# B&R Automation Studio project NAEUL004C00R13L518F00 (part 10)

#### Act_Main_P0933.st
```iecst
ACTION Act_Main_P0933:

	//Display
	tyP0933PushConv.tyFB.tyNumExtSpd.uiRtStat.0			:= NOT p_tyNtParamCurr.bProjMotorizedPusherPrep;
	tyP0933PushConv.tyFB.tyNumExtTorqPercent.uiRtStat.0	:= NOT p_tyNtParamCurr.bProjMotorizedPusherPrep;

	tyP0933PushConv.tyDC.tyBtnSpdBinBit0.uiRtStat.0	:=  NOT p_tyNtParamCurr.bProjMotorizedPusherPrep;
	tyP0933PushConv.tyDC.tyBtnSpdBinBit1.uiRtStat.0	:=  NOT p_tyNtParamCurr.bProjMotorizedPusherPrep;
	tyP0933PushConv.tyDC.tyBtnSpdBinBit2.uiRtStat.0	:=  NOT p_tyNtParamCurr.bProjMotorizedPusherPrep;

	tyP0933PushConv.tyDC.tyBtnSigOn.uiRtStat.0	:=  NOT p_tyNtParamCurr.bProjMotorizedPusherPrep;
	tyP0933PushConv.tyDC.tyBtnAlarmRst.uiRtStat.0:=  NOT p_tyNtParamCurr.bProjMotorizedPusherPrep;

	//Display
	tyP0933PushConv.tyFB.tyNumExtSpd.diValueMin	:= p_tyNtParamCurr.tyProdRcpMtrPshrExtSpd.diMin;
	tyP0933PushConv.tyFB.tyNumExtSpd.diValueMax	:= p_tyNtParamCurr.tyProdRcpMtrPshrExtSpd.diMax;

	tyP0933PushConv.tyFB.tyNumExtTorqPercent.diValueMin	:= p_tyNtParamCurr.tyProdRcpMtrPshrExtTorq.diMin;
	tyP0933PushConv.tyFB.tyNumExtTorqPercent.diValueMax	:= p_tyNtParamCurr.tyProdRcpMtrPshrExtTorq.diMax;

	tyP0933PushConv.tyCom.tyBtnExtSlwSen.uiRtStat.0 := NOT p_tyNtParamCurr.bProjMotorizedPusherPrep;
	tyP0933PushConv.tyCom.tyBtnRetSlwSen.uiRtStat.0 := NOT p_tyNtParamCurr.bProjMotorizedPusherPrep;
	tyP0933PushConv.tyCom.tyBtnAlarmSig.uiRtStat.0 := NOT p_tyNtParamCurr.bProjMotorizedPusherPrep;
	tyP0933PushConv.tyCom.tyBtnTorqueSig.uiRtStat.0 := NOT p_tyNtParamCurr.bProjMotorizedPusherPrep;

	tyP0933PushConv.tyDC.tyBtnAlarmRst.uiRtStat.0 := NOT p_tyNtParamCurr.bProjMotorizedPusherPrep;
	tyP0933PushConv.tyDC.tyBtnSigOn.uiRtStat.0 := NOT p_tyNtParamCurr.bProjMotorizedPusherPrep;

	tyP0933PushConv.tyCom.tyBtnAntiJamSen.uiRtStat.0 := p_tyNtParamCurr.tyDISettings.diPshrAntiJam = 0;
	tyP0933PushConv.tyCom.tyBtnAlarmSig.uiRtStat.0	 := p_tyNtParamCurr.tyDISettings.diMtrPshrAlmSig = 0;
	tyP0933PushConv.tyCom.tyBtnTorqueSig.uiRtStat.0  := p_tyNtParamCurr.tyDISettings.diMtrPshrTorqueSig = 0;

END_ACTION
```

#### Act_Main_P0934.st
```iecst
ACTION Act_Main_P0934:

	//Display
	tyP0934AW.tyMotionStd.tyNumTargetPos.diValue	:= 0;
	tyP0934AW.tyMotionStd.tyNumStepSize.diValue		:= 0;
	tyP0934AW.tyMotionStd.tyNumNomSpd.diValue		:= (p_tyNtParamCurr.tyUIAWNomSpd.diMax + p_tyNtParamCurr.tyUIAWNomSpd.diMin) / 2;
	tyP0934AW.tyMotionStd.tyNumSlwSpd.diValue		:= (p_tyNtParamCurr.tyUIAWSlwSpd.diMax + p_tyNtParamCurr.tyUIAWSlwSpd.diMin) / 3;

	tyP0934AW.tyMotionStd.tyNumTargetPos.diValueMax	:= p_tyNtParamCurr.tyProdRcpWidth.diMax;
	tyP0934AW.tyMotionStd.tyNumTargetPos.diValueMin	:= p_tyNtParamCurr.tyUIAWTargetPos.diMin;

	tyP0934AW.tyMotionStd.tyNumStepSize.diValueMax	:= p_tyNtParamCurr.tyProdRcpWidth.diMax;
	tyP0934AW.tyMotionStd.tyNumStepSize.diValueMin	:= p_tyNtParamCurr.tyProdRcpWidth.diMax * -1;

	tyP0934AW.tyMotionStd.tyNumNomSpd.diValueMax	:= p_tyNtParamCurr.tyUIAWNomSpd.diMax;
	tyP0934AW.tyMotionStd.tyNumNomSpd.diValueMin	:= p_tyNtParamCurr.tyUIAWNomSpd.diMin;

	tyP0934AW.tyMotionStd.tyNumSlwSpd.diValueMax	:= p_tyNtParamCurr.tyUIAWSlwSpd.diMax;
	tyP0934AW.tyMotionStd.tyNumSlwSpd.diValueMin	:= p_tyNtParamCurr.tyUIAWSlwSpd.diMin;

	tyP0934AW.tyAW.tyNumNewWidth.diValueMax			:= p_tyNtParamCurr.tyProdRcpWidth.diMax;
	tyP0934AW.tyAW.tyNumNewWidth.diValueMin			:= p_tyNtParamCurr.tyProdRcpWidth.diMin;

END_ACTION
```

#### Act_Main_P0935.st
```iecst
ACTION Act_Main_P0935:

	tyP0935Lifter.tyLifter.tyBtnGoLaneB.uiRtStat.0	:= NOT p_tyNtParamCurr.bProjLaneBPrep;
	tyP0935Lifter.tyLifter.tyBtnGoLaneA.uiRtStat 		:= p_tyNtParamCurr.bProjMagConvLane1Prep;
	tyP0935Lifter.tyLifter.tyBtnGoLaneA.uiMaskRtStat 	:= p_tyNtParamCurr.bProjMagConvLane1Prep;
	tyP0935Lifter.tyLifter.tyBtnGoLaneD_G.uiRtStat 		:= NOT (p_tyNtParamCurr.bProjMagConvLane1Prep);
	tyP0935Lifter.tyLifter.tyBtnGoLaneD_G.uiMaskRtStat 	:= NOT (p_tyNtParamCurr.bProjMagConvLane1Prep);
	tyP0935Lifter.tyLifter.tyBtnGoLaneE_H.uiRtStat 		:= NOT (p_tyNtParamCurr.bProjMagConvLane1Prep);
	tyP0935Lifter.tyLifter.tyBtnGoLaneE_H.uiMaskRtStat 	:= NOT (p_tyNtParamCurr.bProjMagConvLane1Prep);

	//Display
	tyP0935Lifter.tyMotionStd.tyNumTargetPos.diValue	:= 0;
	tyP0935Lifter.tyMotionStd.tyNumStepSize.diValue		:= 0;
	tyP0935Lifter.tyMotionStd.tyNumNomSpd.diValue		:= (p_tyNtParamCurr.tyUILifterNomSpd.diMax + p_tyNtParamCurr.tyUILifterNomSpd.diMin) / 2;
	tyP0935Lifter.tyMotionStd.tyNumSlwSpd.diValue		:= (p_tyNtParamCurr.tyUILifterSlwSpd.diMax + p_tyNtParamCurr.tyUILifterSlwSpd.diMin) / 3;

	tyP0935Lifter.tyMotionStd.tyNumTargetPos.diValueMax	:= p_tyNtParamCurr.tyUILifterTargetPos.diMax;
	tyP0935Lifter.tyMotionStd.tyNumTargetPos.diValueMin	:= p_tyNtParamCurr.tyUILifterTargetPos.diMin;

	tyP0935Lifter.tyMotionStd.tyNumStepSize.diValueMax	:= p_tyNtParamCurr.tyUILifterStepSize.diMax;
	tyP0935Lifter.tyMotionStd.tyNumStepSize.diValueMin	:= p_tyNtParamCurr.tyUILifterStepSize.diMin;

	tyP0935Lifter.tyMotionStd.tyNumNomSpd.diValueMax	:= p_tyNtParamCurr.tyUILifterNomSpd.diMax;
	tyP0935Lifter.tyMotionStd.tyNumNomSpd.diValueMin	:= p_tyNtParamCurr.tyUILifterNomSpd.diMin;

	tyP0935Lifter.tyMotionStd.tyNumSlwSpd.diValueMax	:= p_tyNtParamCurr.tyUILifterSlwSpd.diMax;
	tyP0935Lifter.tyMotionStd.tyNumSlwSpd.diValueMin	:= p_tyNtParamCurr.tyUILifterSlwSpd.diMin;

	tyP0935Lifter.tyLifter.tyNumMagPos.diValue			:= 1;
	tyP0935Lifter.tyLifter.tyNumMagPos.diValueMin		:= 1;

	CASE p_tyNtParamCurr.eProjMag OF

		ULMagDual:
			IF p_tyNtParamCurr.bProjMagConvLane1Prep THEN
				tyP0935Lifter.tyLifter.tyNumMagPos.diValueMax		:= 1;
			ELSE
				tyP0935Lifter.tyLifter.tyNumMagPos.diValueMax		:= 2;
			END_IF

		ULMagTriple:
			tyP0935Lifter.tyLifter.tyNumMagPos.diValueMax		:= 3;

		ULMagQuadruple:
			tyP0935Lifter.tyLifter.tyNumMagPos.diValueMax		:= 4;

	END_CASE

	IF p_tyNtParamCurr.bProjLifterMagPlatform THEN
		tyP0935Lifter.tyLifter.tyBtnGoLaneA.usiTxtIdx := 23;
	END_IF

END_ACTION
```

#### Act_Main_P0936.st
```iecst
ACTION Act_Main_P0936:

	//Display
	tyP0936Trav.tyTrav.tyBtnGoToLaneB.uiRtStat.0	:= NOT p_tyNtParamCurr.bProjLaneBPrep;
	tyP0936Trav.tyTrav.tyBtnGoToMag3.uiRtStat.0		:= NOT(p_tyNtParamCurr.eProjMag = ULMagTriple);

	tyP0936Trav.tyMotionStd.tyNumTargetPos.diValue		:= 0;
	tyP0936Trav.tyMotionStd.tyNumStepSize.diValue		:= 0;
	tyP0936Trav.tyMotionStd.tyNumNomSpd.diValue			:= (p_tyNtParamCurr.tyUITravNomSpd.diMax + p_tyNtParamCurr.tyUITravNomSpd.diMin) / 2;
	tyP0936Trav.tyMotionStd.tyNumSlwSpd.diValue			:= (p_tyNtParamCurr.tyUITravSlwSpd.diMax + p_tyNtParamCurr.tyUITravSlwSpd.diMin) / 3;

	tyP0936Trav.tyMotionStd.tyNumTargetPos.diValueMax	:= p_tyNtParamCurr.tyUITravTargetPos.diMax;
	tyP0936Trav.tyMotionStd.tyNumTargetPos.diValueMin	:= p_tyNtParamCurr.tyUITravTargetPos.diMin;

	tyP0936Trav.tyMotionStd.tyNumStepSize.diValueMax	:= p_tyNtParamCurr.tyUITravStepSize.diMax;
	tyP0936Trav.tyMotionStd.tyNumStepSize.diValueMin	:= p_tyNtParamCurr.tyUITravStepSize.diMin;

	tyP0936Trav.tyMotionStd.tyNumNomSpd.diValueMax		:= p_tyNtParamCurr.tyUITravNomSpd.diMax;
	tyP0936Trav.tyMotionStd.tyNumNomSpd.diValueMin		:= p_tyNtParamCurr.tyUITravNomSpd.diMin;

	tyP0936Trav.tyMotionStd.tyNumSlwSpd.diValueMax		:= p_tyNtParamCurr.tyUITravSlwSpd.diMax;
	tyP0936Trav.tyMotionStd.tyNumSlwSpd.diValueMin		:= p_tyNtParamCurr.tyUITravSlwSpd.diMin;

END_ACTION
```

#### Act_Main_P0937.st
```iecst
ACTION Act_Main_P0937:

	//Display
	tyP0937AWPushOrPuller.tyMotionStd.tyNumTargetPos.diValue	:= 0;
	tyP0937AWPushOrPuller.tyMotionStd.tyNumStepSize.diValue		:= 0;
	tyP0937AWPushOrPuller.tyMotionStd.tyNumNomSpd.diValue		:= (p_tyNtParamCurr.tyUIAWNomSpd.diMax + p_tyNtParamCurr.tyUIAWNomSpd.diMin) / 2;
	tyP0937AWPushOrPuller.tyMotionStd.tyNumSlwSpd.diValue		:= (p_tyNtParamCurr.tyUIAWSlwSpd.diMax + p_tyNtParamCurr.tyUIAWSlwSpd.diMin) / 3;

	tyP0937AWPushOrPuller.tyMotionStd.tyNumTargetPos.diValueMax	:= p_tyNtParamCurr.tyProdRcpWidth.diMax;
	tyP0937AWPushOrPuller.tyMotionStd.tyNumTargetPos.diValueMin	:= p_tyNtParamCurr.tyUIAWTargetPos.diMin;

	tyP0937AWPushOrPuller.tyMotionStd.tyNumStepSize.diValueMax	:= p_tyNtParamCurr.tyProdRcpWidth.diMax;
	tyP0937AWPushOrPuller.tyMotionStd.tyNumStepSize.diValueMin	:= p_tyNtParamCurr.tyProdRcpWidth.diMax * -1;

	tyP0937AWPushOrPuller.tyMotionStd.tyNumNomSpd.diValueMax	:= p_tyNtParamCurr.tyUIAWNomSpd.diMax;
	tyP0937AWPushOrPuller.tyMotionStd.tyNumNomSpd.diValueMin	:= p_tyNtParamCurr.tyUIAWNomSpd.diMin;

	tyP0937AWPushOrPuller.tyMotionStd.tyNumSlwSpd.diValueMax	:= p_tyNtParamCurr.tyUIAWSlwSpd.diMax;
	tyP0937AWPushOrPuller.tyMotionStd.tyNumSlwSpd.diValueMin	:= p_tyNtParamCurr.tyUIAWSlwSpd.diMin;

	tyP0937AWPushOrPuller.tyAW.tyNumNewWidth.diValueMax			:= p_tyNtParamCurr.tyProdRcpWidth.diMax;
	tyP0937AWPushOrPuller.tyAW.tyNumNewWidth.diValueMin			:= p_tyNtParamCurr.tyProdRcpWidth.diMin;

END_ACTION
```

#### Act_Main_P0938.st
```iecst
ACTION Act_Main_P0938:

	//Display
	//Magazine Auto Width 1
	tyP0938MagAW.tyMotionStd1.tyNumTargetPos.diValue	:= 0;
	tyP0938MagAW.tyMotionStd1.tyNumStepSize.diValue		:= 0;
	tyP0938MagAW.tyMotionStd1.tyNumNomSpd.diValue		:= (p_tyNtParamCurr.tyUIMagAWNomSpd.diMax + p_tyNtParamCurr.tyUIMagAWNomSpd.diMin) / 2;
	tyP0938MagAW.tyMotionStd1.tyNumSlwSpd.diValue		:= (p_tyNtParamCurr.tyUIMagAWSlwSpd.diMax + p_tyNtParamCurr.tyUIMagAWSlwSpd.diMin) / 3;

	tyP0938MagAW.tyMotionStd1.tyNumTargetPos.diValueMax	:= p_tyNtParamCurr.tyProdRcpWidth.diMax;
	tyP0938MagAW.tyMotionStd1.tyNumTargetPos.diValueMin	:= p_tyNtParamCurr.tyUIMagAWTargetPos.diMin;

	tyP0938MagAW.tyMotionStd1.tyNumStepSize.diValueMax	:= p_tyNtParamCurr.tyProdRcpWidth.diMax;
	tyP0938MagAW.tyMotionStd1.tyNumStepSize.diValueMin	:= p_tyNtParamCurr.tyProdRcpWidth.diMax * -1;

	tyP0938MagAW.tyMotionStd1.tyNumNomSpd.diValueMax	:= p_tyNtParamCurr.tyUIMagAWNomSpd.diMax;
	tyP0938MagAW.tyMotionStd1.tyNumNomSpd.diValueMin	:= p_tyNtParamCurr.tyUIMagAWNomSpd.diMin;

	tyP0938MagAW.tyMotionStd1.tyNumSlwSpd.diValueMax	:= p_tyNtParamCurr.tyUIMagAWSlwSpd.diMax;
	tyP0938MagAW.tyMotionStd1.tyNumSlwSpd.diValueMin	:= p_tyNtParamCurr.tyUIMagAWSlwSpd.diMin;

	tyP0938MagAW.tyMagAW1.tyNumNewWidth.diValueMax		:= p_tyNtParamCurr.tyProdRcpWidth.diMax;
	tyP0938MagAW.tyMagAW1.tyNumNewWidth.diValueMin		:= p_tyNtParamCurr.tyProdRcpWidth.diMin;

	//Magazine Auto Width 2
	tyP0938MagAW.tyMotionStd2.tyNumTargetPos.diValue	:= 0;
	tyP0938MagAW.tyMotionStd2.tyNumStepSize.diValue		:= 0;
	tyP0938MagAW.tyMotionStd2.tyNumNomSpd.diValue		:= (p_tyNtParamCurr.tyUIMagAWNomSpd.diMax + p_tyNtParamCurr.tyUIMagAWNomSpd.diMin) / 2;
	tyP0938MagAW.tyMotionStd2.tyNumSlwSpd.diValue		:= (p_tyNtParamCurr.tyUIMagAWSlwSpd.diMax + p_tyNtParamCurr.tyUIMagAWSlwSpd.diMin) / 3;

	tyP0938MagAW.tyMotionStd2.tyNumTargetPos.diValueMax	:= p_tyNtParamCurr.tyProdRcpWidth.diMax;
	tyP0938MagAW.tyMotionStd2.tyNumTargetPos.diValueMin	:= p_tyNtParamCurr.tyUIMagAWTargetPos.diMin;

	tyP0938MagAW.tyMotionStd2.tyNumStepSize.diValueMax	:= p_tyNtParamCurr.tyProdRcpWidth.diMax;
	tyP0938MagAW.tyMotionStd2.tyNumStepSize.diValueMin	:= p_tyNtParamCurr.tyProdRcpWidth.diMax * -1;

	tyP0938MagAW.tyMotionStd2.tyNumNomSpd.diValueMax	:= p_tyNtParamCurr.tyUIMagAWNomSpd.diMax;
	tyP0938MagAW.tyMotionStd2.tyNumNomSpd.diValueMin	:= p_tyNtParamCurr.tyUIMagAWNomSpd.diMin;

	tyP0938MagAW.tyMotionStd2.tyNumSlwSpd.diValueMax	:= p_tyNtParamCurr.tyUIMagAWSlwSpd.diMax;
	tyP0938MagAW.tyMotionStd2.tyNumSlwSpd.diValueMin	:= p_tyNtParamCurr.tyUIMagAWSlwSpd.diMin;

	tyP0938MagAW.tyMagAW2.tyNumNewWidth.diValueMax		:= p_tyNtParamCurr.tyProdRcpWidth.diMax;
	tyP0938MagAW.tyMagAW2.tyNumNewWidth.diValueMin		:= p_tyNtParamCurr.tyProdRcpWidth.diMin;

	//Magazine Auto Width 3
	tyP0938MagAW.tyMotionStd3.tyNumTargetPos.diValue	:= 0;
	tyP0938MagAW.tyMotionStd3.tyNumStepSize.diValue		:= 0;
	tyP0938MagAW.tyMotionStd3.tyNumNomSpd.diValue		:= (p_tyNtParamCurr.tyUIMagAWNomSpd.diMax + p_tyNtParamCurr.tyUIMagAWNomSpd.diMin) / 2;
	tyP0938MagAW.tyMotionStd3.tyNumSlwSpd.diValue		:= (p_tyNtParamCurr.tyUIMagAWSlwSpd.diMax + p_tyNtParamCurr.tyUIMagAWSlwSpd.diMin) / 3;

	tyP0938MagAW.tyMotionStd3.tyNumTargetPos.diValueMax	:= p_tyNtParamCurr.tyProdRcpWidth.diMax;
	tyP0938MagAW.tyMotionStd3.tyNumTargetPos.diValueMin	:= p_tyNtParamCurr.tyUIMagAWTargetPos.diMin;

	tyP0938MagAW.tyMotionStd3.tyNumStepSize.diValueMax	:= p_tyNtParamCurr.tyProdRcpWidth.diMax;
	tyP0938MagAW.tyMotionStd3.tyNumStepSize.diValueMin	:= p_tyNtParamCurr.tyProdRcpWidth.diMax * -1;

	tyP0938MagAW.tyMotionStd3.tyNumNomSpd.diValueMax	:= p_tyNtParamCurr.tyUIMagAWNomSpd.diMax;
	tyP0938MagAW.tyMotionStd3.tyNumNomSpd.diValueMin	:= p_tyNtParamCurr.tyUIMagAWNomSpd.diMin;

	tyP0938MagAW.tyMotionStd3.tyNumSlwSpd.diValueMax	:= p_tyNtParamCurr.tyUIMagAWSlwSpd.diMax;
	tyP0938MagAW.tyMotionStd3.tyNumSlwSpd.diValueMin	:= p_tyNtParamCurr.tyUIMagAWSlwSpd.diMin;

	tyP0938MagAW.tyMagAW3.tyNumNewWidth.diValueMax		:= p_tyNtParamCurr.tyProdRcpWidth.diMax;
	tyP0938MagAW.tyMagAW3.tyNumNewWidth.diValueMin		:= p_tyNtParamCurr.tyProdRcpWidth.diMin;

END_ACTION
```

#### Act_Main_P0939.st
```iecst
ACTION Act_Main_P0939:

	tyP0939Lifter2.tyLifter.tyBtnGoLaneB.uiRtStat.0	:= NOT p_tyNtParamCurr.bProjLaneBPrep;
	tyP0939Lifter2.tyLifter.tyBtnGoLaneA.uiRtStat.0	:= p_tyNtParamCurr.bProjMagConvLane2Prep;
	tyP0939Lifter2.tyLifter.tyBtnGoLaneA.uiRtStat.0	:= p_tyNtParamCurr.bProjMagConvLane2Prep;
	tyP0935Lifter.tyLifter.tyBtnGoLaneD_G.uiRtStat 		:= NOT (p_tyNtParamCurr.bProjMagConvLane2Prep);
	tyP0935Lifter.tyLifter.tyBtnGoLaneD_G.uiMaskRtStat 	:= NOT (p_tyNtParamCurr.bProjMagConvLane2Prep);
	tyP0935Lifter.tyLifter.tyBtnGoLaneE_H.uiRtStat 		:= NOT (p_tyNtParamCurr.bProjMagConvLane2Prep);
	tyP0935Lifter.tyLifter.tyBtnGoLaneE_H.uiMaskRtStat 	:= NOT (p_tyNtParamCurr.bProjMagConvLane2Prep);

	//Display
	tyP0939Lifter2.tyMotionStd.tyNumTargetPos.diValue	:= 0;
	tyP0939Lifter2.tyMotionStd.tyNumStepSize.diValue		:= 0;
	tyP0939Lifter2.tyMotionStd.tyNumNomSpd.diValue		:= (p_tyNtParamCurr.tyUILifterNomSpd.diMax + p_tyNtParamCurr.tyUILifterNomSpd.diMin) / 2;
	tyP0939Lifter2.tyMotionStd.tyNumSlwSpd.diValue		:= (p_tyNtParamCurr.tyUILifterSlwSpd.diMax + p_tyNtParamCurr.tyUILifterSlwSpd.diMin) / 3;

	tyP0939Lifter2.tyMotionStd.tyNumTargetPos.diValueMax	:= p_tyNtParamCurr.tyUILifterTargetPos.diMax;
	tyP0939Lifter2.tyMotionStd.tyNumTargetPos.diValueMin	:= p_tyNtParamCurr.tyUILifterTargetPos.diMin;

	tyP0939Lifter2.tyMotionStd.tyNumStepSize.diValueMax	:= p_tyNtParamCurr.tyUILifterStepSize.diMax;
	tyP0939Lifter2.tyMotionStd.tyNumStepSize.diValueMin	:= p_tyNtParamCurr.tyUILifterStepSize.diMin;

	tyP0939Lifter2.tyMotionStd.tyNumNomSpd.diValueMax	:= p_tyNtParamCurr.tyUILifterNomSpd.diMax;
	tyP0939Lifter2.tyMotionStd.tyNumNomSpd.diValueMin	:= p_tyNtParamCurr.tyUILifterNomSpd.diMin;

	tyP0939Lifter2.tyMotionStd.tyNumSlwSpd.diValueMax	:= p_tyNtParamCurr.tyUILifterSlwSpd.diMax;
	tyP0939Lifter2.tyMotionStd.tyNumSlwSpd.diValueMin	:= p_tyNtParamCurr.tyUILifterSlwSpd.diMin;

	tyP0939Lifter2.tyLifter.tyNumMagPos.diValue			:= 2;
	tyP0939Lifter2.tyLifter.tyNumMagPos.diValueMin		:= 2;
	tyP0939Lifter2.tyLifter.tyNumMagPos.diValueMax		:= 2;

	CASE p_tyNtParamCurr.eProjMag OF

		ULMagDual:
			tyP0939Lifter2.tyLifter.tyNumMagPos.diValueMax		:= 2;

		ULMagTriple:
			tyP0939Lifter2.tyLifter.tyNumMagPos.diValueMax		:= 3;

		ULMagQuadruple:
			tyP0939Lifter2.tyLifter.tyNumMagPos.diValueMax		:= 4;

	END_CASE

	IF p_tyNtParamCurr.bProjLifterMagPlatform THEN
		tyP0939Lifter2.tyLifter.tyBtnGoLaneA.usiTxtIdx := 23;
	END_IF

END_ACTION
```

#### Act_Main_P0940.st
```iecst
ACTION Act_Main_P0940:

	//Display
	tyP0940CommCtrl.tyUSSMEMAB.tyLyr.uiRtStat.0	:= NOT(p_tyNtParamCurr.bProjLaneBPrep);
	IF p_tyNtParamCurr.bProjAGVPrep AND (p_tyMcParamCurr.eAGVComProtocol <> McSetAGVTCPEnableTCP AND p_tyMcParamCurr.eAGVComProtocol <> McSetAGVTCPDisableTCP) THEN
		tyP0940CommCtrl.tySOT.tySOTLyr1.uiRtStat.0 := FALSE;
		tyP0940CommCtrl.tySOT.tySOTLyr2.uiRtStat.0 := FALSE;
		tyP0940CommCtrl.tySOT.tySOTLyr3.uiRtStat.0 := p_tyNtParamCurr.eProjMag <> ULMagTriple AND p_tyNtParamCurr.eProjMag <> ULMagQuadruple;
		tyP0940CommCtrl.tySOT.tySOTLyr4.uiRtStat.0 := p_tyNtParamCurr.eProjMag <> ULMagQuadruple;
		IF p_tyNtParamCurr.bProjMagConvLane1Prep THEN
			tyP0940CommCtrl.tySOT.tyTxtAIVCommProtocol.uiRtStat.0 := TRUE;
		END_IF
	ELSE

		tyP0940CommCtrl.tySOT.tySOTLyr1.uiRtStat.0 := TRUE;
		tyP0940CommCtrl.tySOT.tySOTLyr2.uiRtStat.0 := TRUE;
		tyP0940CommCtrl.tySOT.tySOTLyr3.uiRtStat.0 := TRUE;
		tyP0940CommCtrl.tySOT.tySOTLyr4.uiRtStat.0 := TRUE;
		IF p_tyNtParamCurr.bProjMagConvLane1Prep THEN
			tyP0940CommCtrl.tySOT.tyTxtAIVCommProtocol.uiRtStat.0 := TRUE;
		END_IF
	END_IF

	tyP0940CommCtrl.tySOT.tyBtnAIVRcv1.uiRtStat.0 := NOT(p_tyNtParamCurr.bProjSOTSensorPrep);
	tyP0940CommCtrl.tySOT.tyBtnAIVRcv2.uiRtStat.0 := NOT(p_tyNtParamCurr.bProjSOTSensorPrep);
	tyP0940CommCtrl.tySOT.tyBtnAIVRcv3.uiRtStat.0 := NOT(p_tyNtParamCurr.bProjSOTSensorPrep);
	tyP0940CommCtrl.tySOT.tyBtnAIVRcv4.uiRtStat.0 := NOT(p_tyNtParamCurr.bProjSOTSensorPrep);

	IF  tyP0940CommCtrl.tySOT.tySOTLyr4.uiRtStat.0 = TRUE AND p_tyNtParamCurr.tyDISettings.diScanComplSig > 0   THEN //if hidden update
		tyP0940CommCtrl.tyDMCRFID.tyLyr.uiRtStat.0 := FALSE;
	ELSE
		tyP0940CommCtrl.tyDMCRFID.tyLyr.uiRtStat.0 := TRUE;
	END_IF
END_ACTION
```

#### Act_Main_P0950.st
```iecst
ACTION Act_Main_P0950:

	//Display
//	tyP0950Simu.tyAGVToMc.tyLyr.uiRtStat.0 := NOT(p_tyNtParamCurr.bProjAGVPrep AND p_tyMcParamCurr.bAGVComEn);
//	tyP0950Simu.tySimu.tyLyr.uiRtStat.0 := TRUE;
	tyP0950Simu.tySimu.tyLyr1.uiRtStat.0 := FALSE ;//NOT(p_tyNtParamCurr.bProjAGVPrep AND p_tyMcParamCurr.bAGVComEn);
	tyP0950Simu.tySimu.tyLyr2.uiRtStat.0 := FALSE ;//NOT(p_tyNtParamCurr.bProjAGVPrep AND p_tyMcParamCurr.bAGVComEn AND p_tyNtParamCurr.eProjMag = ULMagTriple);
	tyP0950Simu.tyAGVToMc.tyLyr.uiRtStat.0 := TRUE ;//NOT(p_tyNtParamCurr.bProjAGVPrep AND p_tyMcParamCurr.bAGVComEn);

	IF p_tyNtParamCurr.eProjMag = ULMagDual THEN
		tyP0950Simu.tyAGVToMc.tyBtnAGV3Occupied.uiRtStat		:= TRUE;
		tyP0950Simu.tyAGVToMc.tyBtnAGVInPos3.uiRtStat   		:= TRUE;
		tyP0950Simu.tyMcToAGV.tyBtnMag3Auto.uiRtStat			:= TRUE;
		tyP0950Simu.tyMcToAGV.tyBtnMag3Empty.uiRtStat   		:= TRUE;
		tyP0950Simu.tyMcToAGV.tyBtnMag3IncorrectModel.uiRtStat 	:= TRUE;
		tyP0950Simu.tyMcToAGV.tyBtnMag3Occupied.uiRtStat 		:= TRUE;
		tyP0950Simu.tyMcToAGV.tyBtnMag3Rdy.uiRtStat				:= TRUE;
	END_IF

END_ACTION
```

#### Act_Main_P1000.st
```iecst
ACTION Act_Main_P1000:

	//P1000 Language
	p_tyMcParamCurr.usiLang	:= 0;

//	fUIInRtStatHide(ADR(tyP1000Lang.tyLang.tyBtnGerman.uiRtStat));
//	fUIInRtStatHide(ADR(tyP1000Lang.tyLang.tyBtnChinese.uiRtStat));

//	tyP1000Lang.tyLang.tyBtnEnglish.bValue				:= FALSE;
//	tyP1000Lang.tyLang.tyBtnEnglish.bRtLk				:= FALSE;
//	tyP1000Lang.tyLang.tyBtnGerman.bValue				:= FALSE;
//	tyP1000Lang.tyLang.tyBtnGerman.bRtLk				:= FALSE;
//	tyP1000Lang.tyLang.tyBtnChinese.bValue				:= FALSE;
//	tyP1000Lang.tyLang.tyBtnChinese.bRtLk				:= FALSE;
//
//	CASE p_tyMcParamCurr.usiLang OF
//		1:
//			tyP1000Lang.tyLang.tyBtnGerman.bValue		:= TRUE;
//			tyP1000Lang.tyLang.tyBtnGerman.bRtLk		:= TRUE;
//		2:
//			tyP1000Lang.tyLang.tyBtnChinese.bValue		:= TRUE;
//			tyP1000Lang.tyLang.tyBtnChinese.bRtLk		:= TRUE;
//		ELSE
//			tyP1000Lang.tyLang.tyBtnEnglish.bValue		:= TRUE;
//			tyP1000Lang.tyLang.tyBtnEnglish.bRtLk		:= TRUE;
//	END_CASE

END_ACTION
```

#### Act_Main_P1020.st
```iecst
ACTION Act_Main_P1020:

	//Display
	tyP1020McSetNavi.tyNavi.tyBtnVCommSet.uiRtStat.0	:= NOT(p_tyNtParamCurr.bLFPrep OR p_tyNtParamCurr.bLCSLFPrep OR p_tyNtParamCurr.bLCSReqRcpPrep OR p_tyNtParamCurr.bLCSLiveDatPrep);
	tyP1020McSetNavi.tyNavi.tyBtnOpConSet.uiRtStat.0	:= NOT(p_tyNtParamCurr.bProjOpConPrep);
	tyP1020McSetNavi.tyNavi.tyBtnScanSet.uiRtStat.0		:= NOT(p_tyNtParamCurr.bProjScanPrep);

	//new for Hermes 1.3
	IF (p_tyNtParamCurr.bHermesSvyPrep AND p_tyMcParamCurr.bHermesSvyEn)
		OR p_tyNtParamCurr.bLFPrep OR p_tyNtParamCurr.bLCSLFPrep OR p_tyNtParamCurr.bLCSReqRcpPrep OR p_tyNtParamCurr.bLCSLiveDatPrep
		OR p_tyNtParamCurr.bLCSManageRcpPrep OR p_tyNtParamCurr.bLFUsrSetPrep OR p_tyNtParamCurr.bLFUsrSetPrep
		OR p_tyNtParamCurr.bUSWidthChkPrep OR p_tyNtParamCurr.bDSWidthChkPrep THEN

		fUIInRtStatOff(ADR(tyP1020McSetNavi.tyNavi.tyBtnVCommSet.uiRtStat));
	ELSE
		fUIInRtStatHide(ADR(tyP1020McSetNavi.tyNavi.tyBtnVCommSet.uiRtStat));
	END_IF
END_ACTION
```

#### Act_Main_P1021.st
```iecst
ACTION Act_Main_P1021:

	 //Machine Setting - General
	tyP1021McSetGen.tyGen.tyNumConvInitTm.diValueMin	:= p_tyNtParamCurr.tyUIConvInitTm.diMin;
	tyP1021McSetGen.tyGen.tyNumConvInitTm.diValueMax	:= p_tyNtParamCurr.tyUIConvInitTm.diMax;

	tyP1021McSetGen.tyGen.tyNumMag1ConvRunTm.diValueMin	:= p_tyNtParamCurr.tyUIMagConvRunTm.diMin;
	tyP1021McSetGen.tyGen.tyNumMag1ConvRunTm.diValueMax	:= p_tyNtParamCurr.tyUIMagConvRunTm.diMax;
	tyP1021McSetGen.tyGen.tyNumMag2ConvRunTm.diValueMin	:= p_tyNtParamCurr.tyUIMagConvRunTm.diMin;
	tyP1021McSetGen.tyGen.tyNumMag2ConvRunTm.diValueMax	:= p_tyNtParamCurr.tyUIMagConvRunTm.diMax;
	tyP1021McSetGen.tyGen.tyNumMag3ConvRunTm.diValueMin	:= p_tyNtParamCurr.tyUIMagConvRunTm.diMin;
	tyP1021McSetGen.tyGen.tyNumMag3ConvRunTm.diValueMax	:= p_tyNtParamCurr.tyUIMagConvRunTm.diMax;

	tyP1021McSetGen.tyGen.tyNumTranInErrDlyTm.diValueMin	:= p_tyNtParamCurr.tyUITranInErrDlyTm.diMin;
	tyP1021McSetGen.tyGen.tyNumTranInErrDlyTm.diValueMax	:= p_tyNtParamCurr.tyUITranInErrDlyTm.diMax;

	tyP1021McSetGen.tyGen.tyNumMag1WidthChkDetDist.diValueMin := -7000;
	tyP1021McSetGen.tyGen.tyNumMag1WidthChkDetDist.diValueMax := 7000;

	tyP1021McSetGen.tyGen.tyNumMag2WidthChkDetDist.diValueMin := -7000;
	tyP1021McSetGen.tyGen.tyNumMag2WidthChkDetDist.diValueMax := 7000;

	tyP1021McSetGen.tyGen.tyNumMag3WidthChkDetDist.diValueMin := -7000;
	tyP1021McSetGen.tyGen.tyNumMag3WidthChkDetDist.diValueMax := 7000;
	//MagConv LifterConv
	tyP1021McSetGen.tyGen.tyNumInMagConvInitTm.diValueMin		:= p_tyNtParamCurr.tyUIMagConvRunTm.diMin; //Lane1
	tyP1021McSetGen.tyGen.tyNumInMagConvInitTm.diValueMax		:= p_tyNtParamCurr.tyUIMagConvRunTm.diMax;
	tyP1021McSetGen.tyGen.tyNumOutMagConvInitTm.diValueMin		:= p_tyNtParamCurr.tyUIMagConvRunTm.diMin;
	tyP1021McSetGen.tyGen.tyNumOutMagConvInitTm.diValueMax		:= p_tyNtParamCurr.tyUIMagConvRunTm.diMax;
	tyP1021McSetGen.tyGen.tyNumLifterMagConvInitTm.diValueMin	:= p_tyNtParamCurr.tyUIMagConvRunTm.diMin;
	tyP1021McSetGen.tyGen.tyNumLifterMagConvInitTm.diValueMax	:= p_tyNtParamCurr.tyUIMagConvRunTm.diMax;

	tyP1021McSetGen.tyGen.tyNumLifterTopPos.diValueMin			:= p_tyNtParamCurr.tyUILifterTopPos.diMin;
	tyP1021McSetGen.tyGen.tyNumLifterTopPos.diValueMax			:= p_tyNtParamCurr.tyUILifterTopPos.diMax;
	tyP1021McSetGen.tyGen.tyNumLifterBtmPos.diValueMin			:= p_tyNtParamCurr.tyUILifterBtmPos.diMin;
	tyP1021McSetGen.tyGen.tyNumLifterBtmPos.diValueMax			:= p_tyNtParamCurr.tyUILifterBtmPos.diMax;

	tyP1021McSetGen.tyGen.tyNumInMagConv2InitTm.diValueMin		:= p_tyNtParamCurr.tyUIMagConvRunTm.diMin; //Lane2
	tyP1021McSetGen.tyGen.tyNumInMagConv2InitTm.diValueMax		:= p_tyNtParamCurr.tyUIMagConvRunTm.diMax;
	tyP1021McSetGen.tyGen.tyNumOutMagConv2InitTm.diValueMin		:= p_tyNtParamCurr.tyUIMagConvRunTm.diMin;
	tyP1021McSetGen.tyGen.tyNumOutMagConv2InitTm.diValueMax		:= p_tyNtParamCurr.tyUIMagConvRunTm.diMax;
	tyP1021McSetGen.tyGen.tyNumLifterMagConv2InitTm.diValueMin	:= p_tyNtParamCurr.tyUIMagConvRunTm.diMin;
	tyP1021McSetGen.tyGen.tyNumLifterMagConv2InitTm.diValueMax	:= p_tyNtParamCurr.tyUIMagConvRunTm.diMax;

	tyP1021McSetGen.tyGen.tyNumLifterTopPos2.diValueMin			:= p_tyNtParamCurr.tyUILifterTopPos.diMin;
	tyP1021McSetGen.tyGen.tyNumLifterTopPos2.diValueMax			:= p_tyNtParamCurr.tyUILifterTopPos.diMax;
	tyP1021McSetGen.tyGen.tyNumLifterBtmPos2.diValueMin			:= p_tyNtParamCurr.tyUILifterBtmPos.diMin;
	tyP1021McSetGen.tyGen.tyNumLifterBtmPos2.diValueMax			:= p_tyNtParamCurr.tyUILifterBtmPos.diMax;
	//Siemen
	tyP1021McSetGen.tyGen.tyNumMESResponseTO.diValueMax		:= 30000; //30s
	tyP1021McSetGen.tyGen.tyNumDMCScanWriteTO.diValueMax		:= 30000; //30s

	//Screen Saver
	tyP1021McSetGen.tyGen.tyNumSSaverTm.diValueMin	:= p_tyNtParamCurr.tyUISSaverTm.diMin;
	tyP1021McSetGen.tyGen.tyNumSSaverTm.diValueMax	:= p_tyNtParamCurr.tyUISSaverTm.diMax;
	tyP1021McSetGen.tyGen.tyNumSSaverTm.uiRtStat.0	:= NOT p_tyNtParamCurr.bSSaverPrep;
	tyP1021McSetGen.tyGen.tyBtnSSaverEn.uiRtStat.0	:= NOT p_tyNtParamCurr.bSSaverPrep;
	tyP1021McSetGen.tyGen.tyTxtLblSSaver.uiRtStat.0	:= NOT p_tyNtParamCurr.bSSaverPrep;

	//Width
	tyP1021McSetGen.tyGen.tyNumWidthAtHm.diValueMin	:= p_tyNtParamCurr.tyProdRcpWidth.diMin;
	tyP1021McSetGen.tyGen.tyNumWidthAtHm.diValueMax	:= p_tyNtParamCurr.tyProdRcpWidth.diMax + 10000;
	tyP1021McSetGen.tyGen.tyNumWidthAtHm.uiRtStat.0	:= NOT p_tyNtParamCurr.bAWPrep;
	tyP1021McSetGen.tyGen.tyTxtWidthAtHm.uiRtStat.0	:= NOT p_tyNtParamCurr.bAWPrep;
	tyP1021McSetGen.tyGen.tyBtnAWDis.uiRtStat.0		:= NOT p_tyNtParamCurr.bAWPrep;

	//	tyP1021McSetGen.tyGen.tyNumWidthOffset.uiRtStat.0 :=  NOT p_tyNtParamCurr.bAWPrep;
	//	tyP1021McSetGen.tyGen.tyTxtWidthOffset.uiRtStat.0 :=  NOT p_tyNtParamCurr.bAWPrep;
	tyP1021McSetGen.tyGen.tyNumWidthOffset.uiRtStat.0 :=  TRUE;
	tyP1021McSetGen.tyGen.tyTxtWidthOffset.uiRtStat.0 :=  TRUE;
	tyP1021McSetGen.tyGen.tyNumWidthOffset.diValueMin :=  p_tyNtParamCurr.tyUIAWOffset.diMin;
	tyP1021McSetGen.tyGen.tyNumWidthOffset.diValueMax :=  p_tyNtParamCurr.tyUIAWOffset.diMax;
	//Hermes Remote Configuration
	tyP1021McSetGen.tyGen.tyBtnHermesRmtEn.uiRtStat.0	:= NOT p_tyNtParamCurr.bHermesRmtPrep;

	//Hermes Supervisory Configuration
	tyP1021McSetGen.tyGen.tyBtnHermesSvyEn.uiRtStat.0		:= NOT p_tyNtParamCurr.bHermesSvyPrep; //new for Hermes 1.3
	tyP1021McSetGen.tyGen.tyBtnHermesSvyEn.bValue			:= p_tyMcParamCurr.bHermesSvyEn;//new for Hermes 1.3

	//Machine Mode
	tyP1021McSetGen.tyGen.tyDrpDnDefaultMcMod.uiRtStat.0 := TRUE;
	IF p_tyNtParamCurr.bProjLaneBPrep THEN
		tyP1021McSetGen.tyGen.tyDrpDnDefaultMcMod.usiValueMaxIdx	:= 8;
	ELSE
		tyP1021McSetGen.tyGen.tyDrpDnDefaultMcMod.usiValueMaxIdx	:= 2;
	END_IF

	//Fix To Fix Rail Machine
	IF p_tyNtParamCurr.bProjLaneBPrep AND p_tyNtParamCurr.bProjUSFixToFixRail THEN
		tyP1021McSetGen.tyGen.tyNumTravFixtoFixPosInlet.uiRtStat.0 := FALSE;
	ELSE
		tyP1021McSetGen.tyGen.tyNumTravFixtoFixPosInlet.uiRtStat.0 := TRUE;
	END_IF

	//OvenInfo
	tyP1021McSetGen.tyGen.tyNumMaxBffr.diValueMin		:= p_tyNtParamCurr.tyUIOvenMaxBffrBtwnMc.diMin;
	tyP1021McSetGen.tyGen.tyNumMaxBffr.diValueMax		:= p_tyNtParamCurr.tyUIOvenMaxBffrBtwnMc.diMax;
	tyP1021McSetGen.tyGen.tyBtnOvenEn.uiRtStat.0		:= NOT p_tyNtParamCurr.bOvenInfoPrep;
	tyP1021McSetGen.tyGen.tyBtnExtdOvenEn.uiRtStat.0	:= NOT(p_tyNtParamCurr.bOvenInfoPrep AND p_tyNtParamCurr.bOvenInfoExtdPrep);
	tyP1021McSetGen.tyGen.tyNumMaxBffr.uiRtStat.0		:= NOT(p_tyNtParamCurr.bOvenInfoPrep AND p_tyNtParamCurr.bOvenInfoExtdPrep);
	tyP1021McSetGen.tyGen.tyTxtMaxBffr.uiRtStat.0		:= NOT(p_tyNtParamCurr.bOvenInfoPrep AND p_tyNtParamCurr.bOvenInfoExtdPrep);

	//Trav & Lifter For Lane B
	tyP1021McSetGen.tyGen.tyNumTravPosLaneA.diValueMin		:= p_tyNtParamCurr.tyUITravTargetPos.diMin;
	tyP1021McSetGen.tyGen.tyNumTravPosLaneA.diValueMax		:= p_tyNtParamCurr.tyUITravTargetPos.diMax;
	tyP1021McSetGen.tyGen.tyNumTravPosLaneB.diValueMin		:= p_tyNtParamCurr.tyUITravTargetPos.diMin;
	tyP1021McSetGen.tyGen.tyNumTravPosLaneB.diValueMax		:= p_tyNtParamCurr.tyUITravTargetPos.diMax;
	tyP1021McSetGen.tyGen.tyNumLiftPosLaneA.diValueMin		:= p_tyNtParamCurr.tyUILifterTargetPos.diMin;
	tyP1021McSetGen.tyGen.tyNumLiftPosLaneA.diValueMax		:= p_tyNtParamCurr.tyUILifterTargetPos.diMax;
	tyP1021McSetGen.tyGen.tyNumLiftPosLaneB.diValueMin		:= p_tyNtParamCurr.tyUILifterTargetPos.diMin;
	tyP1021McSetGen.tyGen.tyNumLiftPosLaneB.diValueMax		:= p_tyNtParamCurr.tyUILifterTargetPos.diMax;
	tyP1021McSetGen.tyGen.tyTxtTravPosLaneB.uiRtStat.0		:= NOT (p_tyNtParamCurr.bProjLaneBPrep AND p_tyNtParamCurr.bProjUSFixToFixRail = FALSE);
	tyP1021McSetGen.tyGen.tyNumTravPosLaneB.uiRtStat.0		:= NOT (p_tyNtParamCurr.bProjLaneBPrep AND p_tyNtParamCurr.bProjUSFixToFixRail = FALSE);
	tyP1021McSetGen.tyGen.tyBtnTravPosBTeach.uiRtStat.0		:= NOT (p_tyNtParamCurr.bProjLaneBPrep AND p_tyNtParamCurr.bProjUSFixToFixRail = FALSE);
	tyP1021McSetGen.tyGen.tyTxtLiftPosLaneB.uiRtStat.0		:= NOT p_tyNtParamCurr.bProjLaneBPrep;
	tyP1021McSetGen.tyGen.tyNumLiftPosLaneB.uiRtStat.0		:= NOT p_tyNtParamCurr.bProjLaneBPrep;
	tyP1021McSetGen.tyGen.tyBtnLiftPosBTeach.uiRtStat.0		:= NOT p_tyNtParamCurr.bProjLaneBPrep;

	//Vitrual SMEMA
	tyP1021McSetGen.tyGen.tyBtnVSMEMAEn.uiRtStat.0	:= NOT p_tyNtParamCurr.bVSMEMAPrep;

	//Machine Setting - Magazine Inlet Sensor Auto Detect Timer
	tyP1021McSetGen.tyGen.tyNumMagAutoDetSenTm.diValueMin	:= p_tyNtParamCurr.tyUIMcParamMagAutoEntSenTm.diMin;
	tyP1021McSetGen.tyGen.tyNumMagAutoDetSenTm.diValueMax	:= p_tyNtParamCurr.tyUIMcParamMagAutoEntSenTm.diMax;

	//Gap Between Board
	tyP1021McSetGen.tyGen.tyBtnGapBetBrdEn.uiRtStat.0	:= TRUE;

	//Long Board
	tyP1021McSetGen.tyGen.tyBtnLongBrdEn.uiRtStat.0	:= NOT p_tyNtParamCurr.bProjLongBrdPrep;

	//Shutter
	tyP1021McSetGen.tyGen.tyBtnInShutterDis.uiRtStat.0	:= NOT p_tyNtParamCurr.bProjInletShutPrep;

	//Stopper
	tyP1021McSetGen.tyGen.tyBtnStopperADis.uiRtStat.0	:= NOT p_tyNtParamCurr.bProjStopperAPrep;
	tyP1021McSetGen.tyGen.tyBtnStopperBDis.uiRtStat.0	:= NOT p_tyNtParamCurr.bProjStopperBPrep;

	//Magazine Conveyor
	tyP1021McSetGen.tyGen.tyNumMag1ConvRunTm.uiRtStat.0		:= NOT ((p_tyNtParamCurr.bProjMag1ConvPrep AND NOT(p_tyNtParamCurr.bProjLifTravMnlLoad)) AND p_tyNtParamCurr.bProjLifterMagPlatform = FALSE);
	tyP1021McSetGen.tyGen.tyTxtMag1ConvRunTm.uiRtStat.0		:= NOT ((p_tyNtParamCurr.bProjMag1ConvPrep AND NOT(p_tyNtParamCurr.bProjLifTravMnlLoad)) AND p_tyNtParamCurr.bProjLifterMagPlatform = FALSE);
	tyP1021McSetGen.tyGen.tyNumMag2ConvRunTm.uiRtStat.0		:= NOT ((p_tyNtParamCurr.bProjMag2ConvPrep AND NOT(p_tyNtParamCurr.bProjLifTravMnlLoad)) AND p_tyNtParamCurr.bProjLifterMagPlatform = FALSE);
	tyP1021McSetGen.tyGen.tyTxtMag2ConvRunTm.uiRtStat.0		:= NOT ((p_tyNtParamCurr.bProjMag2ConvPrep AND NOT(p_tyNtParamCurr.bProjLifTravMnlLoad)) AND p_tyNtParamCurr.bProjLifterMagPlatform = FALSE);
	tyP1021McSetGen.tyGen.tyNumMag3ConvRunTm.uiRtStat.0		:= NOT((p_tyNtParamCurr.bProjMag3ConvPrep AND NOT(p_tyNtParamCurr.bProjLifTravMnlLoad)) AND (p_tyNtParamCurr.eProjMag = ULMagTriple) AND p_tyNtParamCurr.bProjLifterMagPlatform = FALSE);
	tyP1021McSetGen.tyGen.tyTxtMag3ConvRunTm.uiRtStat.0		:= NOT((p_tyNtParamCurr.bProjMag3ConvPrep AND NOT(p_tyNtParamCurr.bProjLifTravMnlLoad)) AND (p_tyNtParamCurr.eProjMag = ULMagTriple) AND p_tyNtParamCurr.bProjLifterMagPlatform = FALSE);

	//Parameter
	tyP1021McSetGen.tyGen.tyStringMcNm.sValue				:= p_tyMcParamCurr.sMcNm;
	tyP1021McSetGen.tyGen.tyDrpDnDefaultMcMod.usiValueIdx	:= p_tyMcParamCurr.usiDefaultMcMod;
	tyP1021McSetGen.tyGen.tyNumSSaverTm.diValue				:= UINT_TO_DINT(p_tyMcParamCurr.uiSSaverTmInSec);
	tyP1021McSetGen.tyGen.tyBtnSSaverEn.bValue				:= p_tyMcParamCurr.bSSaverEn;
	tyP1021McSetGen.tyGen.tyStringIPAddr.sValue				:= p_sHWInfoIPAddr;
	tyP1021McSetGen.tyGen.tyStringSubnetMask.sValue			:= p_sHWInfoSubnetMask;
	tyP1021McSetGen.tyGen.tyStringHMIIPAddr.sValue			:= p_tyMcParamCurr.sHMIIPAddr;
	tyP1021McSetGen.tyGen.tyNumWidthAtHm.diValue			:= p_tyMcParamCurr.diWidthAtHmPosInUM;
	tyP1021McSetGen.tyGen.tyNumConvInitTm.diValue			:= p_tyMcParamCurr.diConvInitTmInMS;
	tyP1021McSetGen.tyGen.tyNumTranInErrDlyTm.diValue		:= p_tyMcParamCurr.diTranInErrDlyTmInMS;
	tyP1021McSetGen.tyGen.tyNumMag1ConvRunTm.diValue		:= p_tyMcParamCurr.diMag1ConvRunTmOutInMS;
	tyP1021McSetGen.tyGen.tyNumMag2ConvRunTm.diValue		:= p_tyMcParamCurr.diMag2ConvRunTmOutInMS;
	tyP1021McSetGen.tyGen.tyNumMag3ConvRunTm.diValue		:= p_tyMcParamCurr.diMag3ConvRunTmOutInMS;
	tyP1021McSetGen.tyGen.tyNumMaxBffr.diValue				:= p_tyMcParamCurr.diOvenMaxBffr;
	tyP1021McSetGen.tyGen.tyNumMagAutoDetSenTm.diValue		:= p_tyMcParamCurr.diMagAutoDetectSenTmInMS;
	tyP1021McSetGen.tyGen.tyNumMag1WidthAtHm.diValue		:= p_tyMcParamCurr.diMag1WidthAtHmPosInUM;
	tyP1021McSetGen.tyGen.tyNumMag2WidthAtHm.diValue		:= p_tyMcParamCurr.diMag2WidthAtHmPosInUM;
	tyP1021McSetGen.tyGen.tyNumMag3WidthAtHm.diValue		:= p_tyMcParamCurr.diMag3WidthAtHmPosInUM;

	tyP1021McSetGen.tyGen.tyNumTravPosLaneA.diValue			:= p_tyMcParamCurr.diTravPosA;
	tyP1021McSetGen.tyGen.tyNumLiftPosLaneA.diValue			:= p_tyMcParamCurr.diLifterPosA;
	tyP1021McSetGen.tyGen.tyNumTravPosLaneB.diValue			:= p_tyMcParamCurr.diTravPosB;
	tyP1021McSetGen.tyGen.tyNumLiftPosLaneB.diValue			:= p_tyMcParamCurr.diLifterPosB;
	tyP1021McSetGen.tyGen.tyBtnAWDis.bValue					:= p_tyMcParamCurr.bAWDis;
	tyP1021McSetGen.tyGen.tyBtnMnlAccDat.bValue				:= p_tyMcParamCurr.bMnlAccDat;
	tyP1021McSetGen.tyGen.tyBtnAutoStepEn.bValue			:= p_tyMcParamCurr.bAutoStepEn;
	tyP1021McSetGen.tyGen.tyBtnVSMEMAEn.bValue				:= p_tyMcParamCurr.bVSMEMAEn;
	tyP1021McSetGen.tyGen.tyBtnHermesRmtEn.bValue			:= p_tyMcParamCurr.bHermesRmtEn;
	tyP1021McSetGen.tyGen.tyBtnGapBetBrdEn.bValue			:= p_tyMcParamCurr.bGapBwtnBrdEn;
	tyP1021McSetGen.tyGen.tyBtnLongBrdEn.bValue				:= p_tyMcParamCurr.bLongBrdEn;
	tyP1021McSetGen.tyGen.tyBtnOvenEn.bValue				:= p_tyMcParamCurr.bOvenEn;
	tyP1021McSetGen.tyGen.tyBtnExtdOvenEn.bValue			:= p_tyMcParamCurr.bExtdOvenEn;
	tyP1021McSetGen.tyGen.tyBtnInShutterDis.bValue			:= p_tyMcParamCurr.bInShutterDis;
	tyP1021McSetGen.tyGen.tyBtnChgParamEn.bValue			:= p_tyMcParamCurr.bChgParamEn;
	tyP1021McSetGen.tyGen.tyBtnStopperADis.bValue			:= p_tyMcParamCurr.bStopperADis;
	tyP1021McSetGen.tyGen.tyBtnStopperBDis.bValue			:= p_tyMcParamCurr.bStopperBDis;
	tyP1021McSetGen.tyGen.tyBtnAGVComEn.bValue				:= p_tyMcParamCurr.bAGVComEn;
	tyP1021McSetGen.tyGen.tyNumAWPusherAtHm.diValue			:= p_tyMcParamCurr.diAWPusherAtHmPosInUM;

	tyP1021McSetGen.tyGen.tyBtnAWPusherDis.bValue			:= p_tyMcParamCurr.bAWPusherDis;
	tyP1021McSetGen.tyGen.tyBtnMagWidthChkDis.bValue		:= p_tyMcParamCurr.bMagWidthChkDis;

	//Parameter Page3 : MagConv
	tyP1021McSetGen.tyGen.tyNumInMagConvInitTm.diValue			:= p_tyMcParamCurr.diInMagConvRunTmOutInMS; //Lane1
	tyP1021McSetGen.tyGen.tyNumLifterMagConvInitTm.diValue		:= p_tyMcParamCurr.diLifterMagConvRunTmOutInMS;
	tyP1021McSetGen.tyGen.tyNumOutMagConvInitTm.diValue			:= p_tyMcParamCurr.diOutMagConvRunTmOutInMS;
	tyP1021McSetGen.tyGen.tyNumLifterTopPos.diValue				:= p_tyMcParamCurr.diLifterTopPos;
	tyP1021McSetGen.tyGen.tyNumLifterBtmPos.diValue				:= p_tyMcParamCurr.diLifterBtmPos;
	tyP1021McSetGen.tyGen.tyNumInMagConv2InitTm.diValue			:= p_tyMcParamCurr.diInMagConv2RunTmOutInMS; //Lane2
	tyP1021McSetGen.tyGen.tyNumLifterMagConv2InitTm.diValue		:= p_tyMcParamCurr.diLifterMagConv2RunTmOutInMS;
	tyP1021McSetGen.tyGen.tyNumOutMagConv2InitTm.diValue		:= p_tyMcParamCurr.diOutMagConv2RunTmOutInMS;
	tyP1021McSetGen.tyGen.tyNumLifterTopPos2.diValue			:= p_tyMcParamCurr.diLifterTopPos2;
	tyP1021McSetGen.tyGen.tyNumLifterBtmPos2.diValue			:= p_tyMcParamCurr.diLifterBtmPos2;
	tyP1021McSetGen.tyGen.tyNumMag1WidthChkDetDist.diValue		:= p_tyMcParamCurr.diMag1WidthChkDetDist;
	tyP1021McSetGen.tyGen.tyNumMag2WidthChkDetDist.diValue		:= p_tyMcParamCurr.diMag2WidthChkDetDist;
	tyP1021McSetGen.tyGen.tyNumMag3WidthChkDetDist.diValue		:= p_tyMcParamCurr.diMag3WidthChkDetDist;

	//Page 4 :
	//Siemen
	tyP1021McSetGen.tyGen.tyNumMESResponseTO.diValue			:= p_tyMcParamCurr.diMESResponseTOTmInMS; //RFID Write
	tyP1021McSetGen.tyGen.tyBtnInletStopperDis.bValue			:= p_tyMcParamCurr.bInStopperDis;  //Stopper Inlet
	tyP1021McSetGen.tyGen.tyBtnMESEn.bValue					:= p_tyMcParamCurr.bMESEn;	//RFID
	tyP1021McSetGen.tyGen.tyBtnSwitchingProductType.bValue				:= p_tyMcParamCurr.bSwitchingProdType; //AutoRcp
	tyP1021McSetGen.tyGen.tyBtnBatchIDChgOverCmp.bValue				:= p_tyMcParamCurr.bBatchIDChgOverCmp; //AutoRcp
	tyP1021McSetGen.tyGen.tyBtnIgnoreTopClearance.bValue				:= p_tyMcParamCurr.bIgnoreTopClearance; //AutoRcp
	tyP1021McSetGen.tyGen.tyBtnIgnoreBottomClearance.bValue				:= p_tyMcParamCurr.bIgnoreBtmClearance; //AutoRcp
	tyP1021McSetGen.tyGen.tyBtnIgnoreThickness.bValue				:= p_tyMcParamCurr.bIgnoreThickness; //AutoRcp

	//Parameter P1025 : scanner
	tyP1025McSetScan.tyScan.tyBtnTopScanEn.bValue	:= p_tyMcParamCurr.bTopScannerEn;
	tyP1025McSetScan.tyScan.tyBtnBtmScanEn.bValue	:= p_tyMcParamCurr.bBtmScannerEn;
	tyP1025McSetScan.tyScan.tyStringTopScanSvrIP.sValue	:= p_tyMcParamCurr.sTopScanIPAddr;
	tyP1025McSetScan.tyScan.tyNumTopScanSvrPort.diValue	:= p_tyMcParamCurr.uiTopScanSvrPort;
	tyP1025McSetScan.tyScan.tyStringBtmScanSvrIP.sValue	:= p_tyMcParamCurr.sBtmScanIPAddr;
	tyP1025McSetScan.tyScan.tyNumBtmScanSvrPort.diValue	:= p_tyMcParamCurr.uiBtmScanSvrPort;

	//Logout
	tyP1021McSetGen.tyGen.tyNumAutoLogoutTm.diValueMin			:= p_tyNtParamCurr.tyUIAutoLogoutTm.diMin;
	tyP1021McSetGen.tyGen.tyNumAutoLogoutTm.diValueMax			:= p_tyNtParamCurr.tyUIAutoLogoutTm.diMax;
	tyP1021McSetGen.tyGen.tyNumAutoLogoutTm.uiRtStat.0			:= NOT p_tyNtParamCurr.bAutoLogoutPrep;
	tyP1021McSetGen.tyGen.tyBtnAutoLogoutEn.uiRtStat.0			:= NOT p_tyNtParamCurr.bAutoLogoutPrep;
	tyP1021McSetGen.tyGen.tyTxtLblAutoLogoutTm.uiRtStat.0		:= NOT p_tyNtParamCurr.bAutoLogoutPrep;

	tyP1021McSetGen.tyGen.tyNumAutoLogoutTm.diValue				:= p_tyMcParamCurr.diAutoLogoutTmInSec;
	tyP1021McSetGen.tyGen.tyBtnAutoLogoutEn.bValue				:= p_tyMcParamCurr.bAutoLogoutEn;

	//Network Mode
	tyP1021McSetGen.tyGen.tyDrpDnNetworkMod.usiValueMinIdx		:= DINT_TO_USINT(p_tyNtParamCurr.tyNetworkMode.diMin);
	tyP1021McSetGen.tyGen.tyDrpDnNetworkMod.usiValueMaxIdx		:= DINT_TO_USINT(p_tyNtParamCurr.tyNetworkMode.diMax);
	tyP1021McSetGen.tyGen.tyDrpDnNetworkMod.usiValueIdx			:= DINT_TO_USINT(p_tyMcParamCurr.eNetworkMod);

	//Pusher Auto Width AT Home
	tyP1021McSetGen.tyGen.tyNumAWPusherAtHm.diValueMin	:= p_tyNtParamCurr.tyProdRcpWidth.diMin-p_tyNtParamCurr.tyProdRcpWidth.diMin;
	tyP1021McSetGen.tyGen.tyNumAWPusherAtHm.diValueMax	:= (p_tyNtParamCurr.tyProdRcpWidth.diMax + 10000) / 2;
	tyP1021McSetGen.tyGen.tyNumAWPusherAtHm.uiRtStat.0	:= NOT p_tyNtParamCurr.bAWPusherPrep;
	tyP1021McSetGen.tyGen.tyTxtAWPusherAtHm.uiRtStat.0	:= NOT p_tyNtParamCurr.bAWPusherPrep;
	tyP1021McSetGen.tyGen.tyBtnAWPusherDis.uiRtStat.0	:= NOT p_tyNtParamCurr.bAWPusherPrep;

	//Magazine Width
	tyP1021McSetGen.tyGen.tyNumMag1WidthAtHm.diValueMin	:= p_tyNtParamCurr.tyProdRcpWidth.diMin - 10000;
	tyP1021McSetGen.tyGen.tyNumMag1WidthAtHm.diValueMax	:= p_tyNtParamCurr.tyProdRcpWidth.diMax + 10000;
	tyP1021McSetGen.tyGen.tyNumMag2WidthAtHm.diValueMin	:= p_tyNtParamCurr.tyProdRcpWidth.diMin - 10000;
	tyP1021McSetGen.tyGen.tyNumMag2WidthAtHm.diValueMax	:= p_tyNtParamCurr.tyProdRcpWidth.diMax + 10000;
	tyP1021McSetGen.tyGen.tyNumMag3WidthAtHm.diValueMin	:= p_tyNtParamCurr.tyProdRcpWidth.diMin - 10000;
	tyP1021McSetGen.tyGen.tyNumMag3WidthAtHm.diValueMax	:= p_tyNtParamCurr.tyProdRcpWidth.diMax + 10000;
	tyP1021McSetGen.tyGen.tyNumMag1WidthAtHm.uiRtStat.0	:= NOT p_tyNtParamCurr.bProjMagAWPrep;
	tyP1021McSetGen.tyGen.tyTxtMag1WidthAtHm.uiRtStat.0	:= NOT p_tyNtParamCurr.bProjMagAWPrep;
	tyP1021McSetGen.tyGen.tyNumMag2WidthAtHm.uiRtStat.0	:= NOT p_tyNtParamCurr.bProjMagAWPrep;
	tyP1021McSetGen.tyGen.tyTxtMag2WidthAtHm.uiRtStat.0	:= NOT p_tyNtParamCurr.bProjMagAWPrep;
	tyP1021McSetGen.tyGen.tyNumMag3WidthAtHm.uiRtStat.0	:= NOT(p_tyNtParamCurr.bProjMagAWPrep AND p_tyNtParamCurr.eProjMag = ULMagTriple);
	tyP1021McSetGen.tyGen.tyTxtMag3WidthAtHm.uiRtStat.0	:= NOT(p_tyNtParamCurr.bProjMagAWPrep AND p_tyNtParamCurr.eProjMag = ULMagTriple);

	tyP1021McSetGen.tyGen.tyBtnAutoStepEn.uiRtStat.0			:= TRUE;
	//Magazine Wall Auto Width
	tyP1021McSetGen.tyGen.tyBtnMagAWDis.uiRtStat	:= NOT p_tyNtParamCurr.bProjMagAWPrep;
	tyP1021McSetGen.tyGen.tyBtnMagAWDis.bValue				:= p_tyMcParamCurr.bMagAWDis;
	//Magazine Safety Bar
	tyP1021McSetGen.tyGen.tyBtnMagSafetyBarDis.uiRtStat	:= NOT p_tyNtParamCurr.bProjMagSafetyBarPrep;
	tyP1021McSetGen.tyGen.tyBtnMagSafetyBarDis.bValue		:= p_tyMcParamCurr.bMagSafetyBarDis;

	tyP1021McSetGen.tyGen.tyBtnLFBuzMute.bValue				:= p_tyMcParamCurr.bLFBuzMute;

	tyP1021McSetGen.tyGen.tyNumTCPSvrPort.uiRtStat		:= NOT p_tyNtParamCurr.bProjTCPAGVSigPrep;
	tyP1021McSetGen.tyGen.tyNumTCPSvrPort.diValue		:= p_tyMcParamCurr.diTCPSvrPort;

	IF p_tyNtParamCurr.bProjMagConvLane1Prep THEN
		tyP1021McSetGen.tyGen.tyDrpDnAGVComProtocol.usiValueMaxIdx		:= 4;
		tyP1021McSetGen.tyGen.tyDrpDnAGVComProtocol.usiValueMinIdx		:= 3;
	ELSE
		tyP1021McSetGen.tyGen.tyDrpDnAGVComProtocol.usiValueMaxIdx		:= 2;
		tyP1021McSetGen.tyGen.tyDrpDnAGVComProtocol.usiValueMinIdx		:= 0;
	END_IF

	CASE  p_tyMcParamCurr.eAGVComProtocol OF
		McSetAGVCommOPCUA:
			tyP1021McSetGen.tyGen.tyDrpDnAGVComProtocol.usiValueIdx :=  0;

		McSetAGVCommHardIO:
			tyP1021McSetGen.tyGen.tyDrpDnAGVComProtocol.usiValueIdx :=  1;

		McSetAGVCommDisabled:
			tyP1021McSetGen.tyGen.tyDrpDnAGVComProtocol.usiValueIdx :=  2;

		McSetAGVTCPEnableTCP:
			tyP1021McSetGen.tyGen.tyDrpDnAGVComProtocol.usiValueIdx :=  3;
		McSetAGVTCPDisableTCP:
			tyP1021McSetGen.tyGen.tyDrpDnAGVComProtocol.usiValueIdx :=  4;
	END_CASE

	IF p_tyNtParamCurr.bProjAIVInPosSenPrep THEN
		tyP1021McSetGen.tyGen.tyDrpDnMagExchangeMode.usiValueMaxIdx		:= 3;
		tyP1021McSetGen.tyGen.tyDrpDnMagExchangeMode.usiValueMinIdx		:= 4;
	ELSE
		tyP1021McSetGen.tyGen.tyDrpDnMagExchangeMode.usiValueMaxIdx		:= 2;
		tyP1021McSetGen.tyGen.tyDrpDnMagExchangeMode.usiValueMinIdx		:= 0;
	END_IF

	CASE  p_tyMcParamCurr.eMagExMode OF
		McSetMagXcAutoManMode:
			tyP1021McSetGen.tyGen.tyDrpDnMagExchangeMode.usiValueIdx := 0;

		McSetMagXcAutoMode:
			tyP1021McSetGen.tyGen.tyDrpDnMagExchangeMode.usiValueIdx := 1;

		McSetMagXcManMode:
			tyP1021McSetGen.tyGen.tyDrpDnMagExchangeMode.usiValueIdx := 2;
	END_CASE

	tyP1021McSetGen.tyGen.tyDrpDnAGVComProtocol.uiRtStat.0 := NOT p_tyNtParamCurr.bProjAGVPrep;
	tyP1021McSetGen.tyGen.tyDrpDnMagExchangeMode.uiRtStat.0 := NOT p_tyNtParamCurr.bProjAGVPrep;

	tyP1021McSetGen.tyGen.tyBtnAGVComEn.uiRtStat.0 := TRUE;
	tyP1021McSetGen.tyGen.tyBtnAGVSizeDisabled.bValue := p_tyMcParamCurr.bAIVSizeDisabled;

	tyP1021McSetGen.tyGen.tyNumTravFixtoFixPosInlet.diValue		:= p_tyMcParamCurr.diTravInletFixtoFixPos;
	tyP1021McSetGen.tyGen.tyNumTravFixtoFixPosInlet.diValueMax	:= 1000000;

	tyP1021McSetGen.tyGen.tyBtnDisableFMWarning.uiRtStat.0 := NOT((p_tyNtParamCurr.bProjAGVPrep)AND NOT(p_tyNtParamCurr.bProjTCPAGVSigPrep));
	tyP1021McSetGen.tyGen.tyBtnDisableFMWarning.bValue	:= p_tyMcParamCurr.bDisableFMWarning;

	IF p_tyNtParamCurr.bProjLifterMagPlatform THEN
		tyP1021McSetGen.tyGen.tyTxtLiftPosLaneA.usiValueIdx := 23;
	END_IF

	tyP1021McSetGen.tyGen.tyNumMagAutoDetSenTm.uiRtStat.0 := NOT (p_tyNtParamCurr.bProjMag1ConvPrep AND p_tyNtParamCurr.bProjMag2ConvPrep AND p_tyNtParamCurr.bProjMag3ConvPrep AND p_tyNtParamCurr.bProjLifterMagPlatform = FALSE);
	tyP1021McSetGen.tyGen.tyBtnAGVSizeDisabled.uiRtStat.0 := NOT(p_tyNtParamCurr.bProjAGVPrep AND NOT(p_tyNtParamCurr.bProjTCPAGVSigPrep));
	tyP1021McSetGen.tyGen.tyTxtLiftPosLaneA.uiRtStat.0	:= p_tyNtParamCurr.bProjMagConvLane1Prep;
	tyP1021McSetGen.tyGen.tyNumLiftPosLaneA.uiRtStat.0	:= p_tyNtParamCurr.bProjMagConvLane1Prep;
	tyP1021McSetGen.tyGen.tyBtnLiftPosATeach.uiRtStat	:= p_tyNtParamCurr.bProjMagConvLane1Prep;

	//DataSource.UI.UI.p_tyP1021McSetGen.tyBtnMagWidthChkDis.uiRtStat
	//Magazine Width Check
	tyP1021McSetGen.tyGen.tyBtnMagWidthChkDis.uiRtStat.0 :=  NOT(p_tyNtParamCurr.tyDISettings.diMagWidthChkSen > 0);
	tyP1021McSetGen.tyGen.tyNumMag1WidthChkDetDist.uiRtStat.0 :=  NOT(p_tyNtParamCurr.tyDISettings.diMagWidthChkSen > 0);
	tyP1021McSetGen.tyGen.tyNumMag2WidthChkDetDist.uiRtStat.0 :=  NOT(p_tyNtParamCurr.tyDISettings.diMagWidthChkSen > 0);
	tyP1021McSetGen.tyGen.tyNumMag3WidthChkDetDist.uiRtStat.0 :=  NOT(p_tyNtParamCurr.tyDISettings.diMagWidthChkSen > 0);

	tyP1021McSetGen.tyGen.tyBtnInletStopperDis.uiRtStat.0		:= NOT(p_tyNtParamCurr.bProjInletStopperPrep);
	tyP1021McSetGen.tyGen.tyNumInStprDelayTm.uiRtStat.0		:= NOT(p_tyNtParamCurr.bProjInletStopperPrep);
	tyP1021McSetGen.tyGen.tyNumMESResponseTO.uiRtStat.0		:= NOT(p_tyNtParamCurr.eCustomerReq = Siemens );
	tyP1021McSetGen.tyGen.tyBtnMESEn.uiRtStat.0				:= NOT(p_tyNtParamCurr.eCustomerReq = Siemens OR p_tyNtParamCurr.eCustomerReq = We_Fabricate);
	tyP1021McSetGen.tyGen.tyBtnSwitchingProductType.uiRtStat.0		:= TRUE; // NOT(p_tyNtParamCurr.bAutoRcpPrep);
	tyP1021McSetGen.tyGen.tyBtnBatchIDChgOverCmp.uiRtStat.0		:= NOT(p_tyNtParamCurr.bAutoRcpPrep AND p_tyNtParamCurr.eAutoRcpPrecededBy = PrecededBySelf);

	tyP1021McSetGen.tyGen.tyBtnIgnoreTopClearance.uiRtStat.0	 := NOT(p_tyNtParamCurr.bAutoRcpPrep AND p_tyNtParamCurr.eAutoRcpPrecededBy = PrecededBySelf);
	tyP1021McSetGen.tyGen.tyBtnIgnoreBottomClearance.uiRtStat.0	 := NOT(p_tyNtParamCurr.bAutoRcpPrep AND p_tyNtParamCurr.eAutoRcpPrecededBy = PrecededBySelf);
	tyP1021McSetGen.tyGen.tyBtnIgnoreThickness.uiRtStat.0	 := NOT(p_tyNtParamCurr.bAutoRcpPrep AND p_tyNtParamCurr.eAutoRcpPrecededBy = PrecededBySelf);
	tyP1021McSetGen.tyGen.tyBtnDMCScannerEn.uiRtStat.0  := NOT(p_tyNtParamCurr.tyDISettings.diScanComplSig >0 );
	tyP1021McSetGen.tyGen.tyNumDMCScanWriteTO.uiRtStat.0  := NOT(p_tyNtParamCurr.tyDISettings.diScanComplSig >0 );
	tyP1021McSetGen.tyGen.tyBtnDMCScannerEn.bValue := p_tyMcParamCurr.bDMCScannerEn;
	tyP1021McSetGen.tyGen.tyNumDMCScanWriteTO.diValue := p_tyMcParamCurr.diDMCScanTOErrInMs;

	//Button Position Limit
	tyP1021McSetGen.tyGen.tyDrpDnPos1.usiValueMinIdx			:= DINT_TO_USINT (p_tyNtParamCurr.tyUIBtnPosLmt.diMin);
	tyP1021McSetGen.tyGen.tyDrpDnPos1.usiValueMaxIdx			:= DINT_TO_USINT (p_tyNtParamCurr.tyUIBtnPosLmt.diMax);

	tyP1021McSetGen.tyGen.tyDrpDnPos2.usiValueMinIdx			:= DINT_TO_USINT (p_tyNtParamCurr.tyUIBtnPosLmt.diMin);
	tyP1021McSetGen.tyGen.tyDrpDnPos2.usiValueMaxIdx			:= DINT_TO_USINT (p_tyNtParamCurr.tyUIBtnPosLmt.diMax);

	tyP1021McSetGen.tyGen.tyDrpDnPos3.usiValueMinIdx			:= DINT_TO_USINT (p_tyNtParamCurr.tyUIBtnPosLmt.diMin);
	tyP1021McSetGen.tyGen.tyDrpDnPos3.usiValueMaxIdx			:= DINT_TO_USINT (p_tyNtParamCurr.tyUIBtnPosLmt.diMax);

//	tyP1021McSetGen.tyGen.tyDrpDnPos4.usiValueMinIdx			:= DINT_TO_USINT (p_tyNtParamCurr.tyUIBtnPosLmt.diMin);
//	tyP1021McSetGen.tyGen.tyDrpDnPos4.usiValueMaxIdx			:= DINT_TO_USINT (p_tyNtParamCurr.tyUIBtnPosLmt.diMax);

	tyP1021McSetGen.tyGen.tyDrpDnPos1.uiRtStat.0			:= TRUE; //buzzer no required
	tyP1021McSetGen.tyGen.tyDrpDnPos2.uiRtStat.0			:= TRUE;
	tyP1021McSetGen.tyGen.tyDrpDnPos3.uiRtStat.0			:= TRUE;
//	tyP1021McSetGen.tyGen.tyDrpDnPos4.uiRtStat.0			:= FALSE;

	tyP1021McSetGen.tyGen.tyDrpDnPos1.usiValueIdx			:= DINT_TO_USINT (p_tyMcParamCurr.tyOptBtnPos.ePos1);
	tyP1021McSetGen.tyGen.tyDrpDnPos2.usiValueIdx			:= DINT_TO_USINT (p_tyMcParamCurr.tyOptBtnPos.ePos2);
	tyP1021McSetGen.tyGen.tyDrpDnPos3.usiValueIdx			:= DINT_TO_USINT (p_tyMcParamCurr.tyOptBtnPos.ePos3);

	tyP1021McSetGen.tyGen.tyStringDefaultGWIP.sValue			:= p_tyMcParamCurr.sDefaultGateWay;
END_ACTION
```

#### Act_Main_P1022.st
```iecst
ACTION Act_Main_P1022:

	//Machine Setting - Vertical Communicationm Control
	//Display
	tyP1022McSetVComm.tyVComSel.tyBtnLF.uiRtStat.0				:= NOT p_tyNtParamCurr.bLFPrep;
	tyP1022McSetVComm.tyVComSel.tyBtnLCSLF.uiRtStat.0			:= NOT p_tyNtParamCurr.bLCSLFPrep;
	tyP1022McSetVComm.tyVComSel.tyBtnLCSReqRcp.uiRtStat.0		:= NOT p_tyNtParamCurr.bLCSReqRcpPrep;
	tyP1022McSetVComm.tyVComSel.tyBtnLCSManageRcp.uiRtStat.0	:= NOT p_tyNtParamCurr.bLCSManageRcpPrep;
	tyP1022McSetVComm.tyVComSel.tyBtnLCSLiveDat.uiRtStat.0		:= NOT p_tyNtParamCurr.bLCSLiveDatPrep;

	tyP1022McSetVComm.tyLF.tyBtnLeaderMc.uiRtStat.0			:= NOT p_tyNtParamCurr.bLFUsrSetPrep;
	tyP1022McSetVComm.tyLF.tyBtnSectionLdr.uiRtStat.0		:= NOT (p_tyNtParamCurr.bLFUsrSetPrep OR p_tyNtParamCurr.bLCSLFPrep);
	tyP1022McSetVComm.tyLF.tyBtnUSWidthChkEn.uiRtStat.0		:= NOT p_tyNtParamCurr.bUSWidthChkPrep;
	tyP1022McSetVComm.tyLF.tyBtnDBAOnWOAlign.uiRtStat.0		:= NOT p_tyNtParamCurr.bDSWidthChkPrep;

	//Parameter
	tyP1022McSetVComm.tyVComSel.tyBtnLF.bValue				:= p_tyMcParamCurr.bLFEn;
	tyP1022McSetVComm.tyVComSel.tyBtnLCSLF.bValue			:= p_tyMcParamCurr.bLCSLFEn;
	tyP1022McSetVComm.tyVComSel.tyBtnLCSReqRcp.bValue		:= p_tyMcParamCurr.bLCSReqRcpEn;
	tyP1022McSetVComm.tyVComSel.tyBtnLCSManageRcp.bValue	:= p_tyMcParamCurr.bLCSManageRcpEn;
	tyP1022McSetVComm.tyVComSel.tyBtnLCSLiveDat.bValue		:= p_tyMcParamCurr.bLCSLiveDatEn;

	tyP1022McSetVComm.tyLF.tyBtnLeaderMc.bValue			:= p_tyMcParamCurr.bLFLeaderMc;
	tyP1022McSetVComm.tyLF.tyBtnSectionLdr.bValue		:= p_tyMcParamCurr.bSectionLeader;
	tyP1022McSetVComm.tyLF.tyBtnUSWidthChkEn.bValue		:= p_tyMcParamCurr.bUSWidthChkEn;
	tyP1022McSetVComm.tyLF.tyBtnDBAOnWOAlign.bValue		:= p_tyMcParamCurr.bDBAOnWOAlign;

	//new for Hermes 1.3
	tyP1022McSetVComm.tyVComSvy.tyNumSndAliveTm.diValue	    	    := TIME_TO_DINT(p_tyHermesConfiguration.tySvyParam.tSndAlive);
	tyP1022McSetVComm.tyVComSvy.tyNumSvySystemPort.diValue	    	:= UINT_TO_DINT(p_tyHermesConfiguration.tySvyParam.uiSvySvstemPort);
	tyP1022McSetVComm.tyVComSvy.tyBtnConfiguration.bValue		    := p_tyHermesConfiguration.tySvyParam.bFeatureConfiguration;
	tyP1022McSetVComm.tyVComSvy.tyBtnCheckAliveResponse.bValue		:= p_tyHermesConfiguration.tySvyParam.bFeatureCheckAliveResponse;
	tyP1022McSetVComm.tyVComSvy.tyBtnBoardTracking.bValue		    := p_tyHermesConfiguration.tySvyParam.bFeatureBoardTracking;
	tyP1022McSetVComm.tyVComSvy.tyBtnQueryWorkOrderInfo.bValue		:= p_tyHermesConfiguration.tySvyParam.bFeatureQueryWorkOrderInfo;
	tyP1022McSetVComm.tyVComSvy.tyBtnSendWorkOrderInfo.bValue		:= p_tyHermesConfiguration.tySvyParam.bFeatureSendWorkOrderInfo;

END_ACTION
```

#### Act_Main_P1023.st
```iecst
ACTION Act_Main_P1023:

	//Machine Setting - Horizontal Communicationm Control
	//Display
	tyP1023McSetHComm.tyUSSelA.tyBtnHermes.uiRtStat.0	:= NOT p_tyNtParamCurr.bHermesPrep;
	tyP1023McSetHComm.tyUSSelB.tyBtnHermes.uiRtStat.0	:= NOT p_tyNtParamCurr.bHermesPrep;

	IF p_tyNtParamCurr.bIPCSMEMA9851ExtdPrep = TRUE THEN
		tyP1023McSetHComm.tyUSSMEMAA.tyDrpDnSMEMAMod.usiValueMaxIdx	:= 2;
		tyP1023McSetHComm.tyUSSMEMAB.tyDrpDnSMEMAMod.usiValueMaxIdx	:= 2;
	ELSE
		tyP1023McSetHComm.tyUSSMEMAA.tyDrpDnSMEMAMod.usiValueMaxIdx	:= 1;
		tyP1023McSetHComm.tyUSSMEMAB.tyDrpDnSMEMAMod.usiValueMaxIdx	:= 1;
	END_IF

	tyP1023McSetHComm.tyUSHermesA.tyNumSndAliveTm.diValueMin	:= p_tyNtParamCurr.tyUIHermesSndAliveTm.diMin;
	tyP1023McSetHComm.tyUSHermesA.tyNumSndAliveTm.diValueMax	:= p_tyNtParamCurr.tyUIHermesSndAliveTm.diMax;
	tyP1023McSetHComm.tyUSHermesB.tyNumSndAliveTm.diValueMin	:= p_tyNtParamCurr.tyUIHermesSndAliveTm.diMin;
	tyP1023McSetHComm.tyUSHermesB.tyNumSndAliveTm.diValueMax	:= p_tyNtParamCurr.tyUIHermesSndAliveTm.diMax;

	tyP1023McSetHComm.tyUSHermesA.tyNumLaneID.diValueMin		:= p_tyNtParamCurr.tyUIHermesLnID.diMin;
	tyP1023McSetHComm.tyUSHermesA.tyNumLaneID.diValueMax		:= p_tyNtParamCurr.tyUIHermesLnID.diMax;
	tyP1023McSetHComm.tyUSHermesB.tyNumLaneID.diValueMin		:= p_tyNtParamCurr.tyUIHermesLnID.diMin;
	tyP1023McSetHComm.tyUSHermesB.tyNumLaneID.diValueMax		:= p_tyNtParamCurr.tyUIHermesLnID.diMax;

	//Parameter - Upstream A
	CASE p_tyMcParamCurr.eUSCommA OF
		McSetCommModSMEMA:
			tyP1023McSetHComm.tyUSSelA.tyBtnSMEMA.bValue	:= TRUE;
			tyP1023McSetHComm.tyUSSelA.tyBtnSMEMA.bRtLk		:= TRUE;
			tyP1023McSetHComm.tyUSSelA.tyBtnHermes.bValue	:= FALSE;
			tyP1023McSetHComm.tyUSSelA.tyBtnHermes.bRtLk	:= FALSE;
		McSetCommModHermes:
			tyP1023McSetHComm.tyUSSelA.tyBtnSMEMA.bValue	:= FALSE;
			tyP1023McSetHComm.tyUSSelA.tyBtnSMEMA.bRtLk		:= FALSE;
			tyP1023McSetHComm.tyUSSelA.tyBtnHermes.bValue	:= TRUE;
			tyP1023McSetHComm.tyUSSelA.tyBtnHermes.bRtLk	:= TRUE;
	END_CASE

	tyP1023McSetHComm.tyUSSMEMAA.tyDrpDnSMEMAMod.usiValueIdx		:= UDINT_TO_USINT(p_tyMcParamCurr.tyUSCommASMEMA.eSelection);
	tyP1023McSetHComm.tyUSSMEMAA.tyBtnGdSig.bValue					:= p_tyMcParamCurr.tyUSCommASMEMA.bStatSigSetGd;

	tyP1023McSetHComm.tyUSHermesA.tyNumSndAliveTm.diValue			:= TIME_TO_DINT(p_tyHermesConfiguration.a_tyUSParam[0].tSndAlive);
	tyP1023McSetHComm.tyUSHermesA.tyNumLaneID.diValue				:= INT_TO_DINT(p_tyHermesConfiguration.a_tyUSParam[0].iLaneID);
	tyP1023McSetHComm.tyUSHermesA.tyNumHostPort.diValue				:= UINT_TO_DINT(p_tyHermesConfiguration.a_tyUSParam[0].uiHostPort);
	tyP1023McSetHComm.tyUSHermesA.tyStringHostAddr.sValue			:= p_tyHermesConfiguration.a_tyUSParam[0].sHostAddress;
	tyP1023McSetHComm.tyUSHermesA.tyBtnCheckAliveResponse.bValue	:= p_tyHermesConfiguration.a_tyUSParam[0].bFeatureCheckAliveResponse;
	tyP1023McSetHComm.tyUSHermesA.tyBtnCmpTypeId.bValue				:= p_tyHermesConfiguration.a_tyUSParam[0].bCmpTypeId;
	tyP1023McSetHComm.tyUSHermesA.tyBtnCmpParam.bValue				:= p_tyHermesConfiguration.a_tyUSParam[0].bCmpParam;
	tyP1023McSetHComm.tyUSHermesA.tyBtnOverWrite.bValue				:= p_tyHermesConfiguration.a_tyUSParam[0].bOverwrite;
	tyP1023McSetHComm.tyUSHermesA.tyBtnBoardForecast.bValue		:= p_tyHermesConfiguration.a_tyUSParam[0].bFeatureBoardForecast;//new for Hermes 1.3
	tyP1023McSetHComm.tyUSHermesA.tyBtnQueryBoardInfo.bValue		:= p_tyHermesConfiguration.a_tyUSParam[0].bFeatureQueryBoardInfo;//new for Hermes 1.3

	//Parameter - Upstream B
	CASE p_tyMcParamCurr.eUSCommB OF
		McSetCommModSMEMA:
			tyP1023McSetHComm.tyUSSelB.tyBtnSMEMA.bValue	:= TRUE;
			tyP1023McSetHComm.tyUSSelB.tyBtnSMEMA.bRtLk		:= TRUE;
			tyP1023McSetHComm.tyUSSelB.tyBtnHermes.bValue	:= FALSE;
			tyP1023McSetHComm.tyUSSelB.tyBtnHermes.bRtLk	:= FALSE;
		McSetCommModHermes:
			tyP1023McSetHComm.tyUSSelB.tyBtnSMEMA.bValue	:= FALSE;
			tyP1023McSetHComm.tyUSSelB.tyBtnSMEMA.bRtLk		:= FALSE;
			tyP1023McSetHComm.tyUSSelB.tyBtnHermes.bValue	:= TRUE;
			tyP1023McSetHComm.tyUSSelB.tyBtnHermes.bRtLk	:= TRUE;
	END_CASE

	tyP1023McSetHComm.tyUSSMEMAB.tyDrpDnSMEMAMod.usiValueIdx		:= UDINT_TO_USINT(p_tyMcParamCurr.tyUSCommBSMEMA.eSelection);
	tyP1023McSetHComm.tyUSSMEMAB.tyBtnGdSig.bValue					:= p_tyMcParamCurr.tyUSCommBSMEMA.bStatSigSetGd;

	tyP1023McSetHComm.tyUSHermesB.tyNumSndAliveTm.diValue			:= TIME_TO_DINT(p_tyHermesConfiguration.a_tyUSParam[1].tSndAlive);
	tyP1023McSetHComm.tyUSHermesB.tyNumLaneID.diValue				:= INT_TO_DINT(p_tyHermesConfiguration.a_tyUSParam[1].iLaneID);
	tyP1023McSetHComm.tyUSHermesB.tyNumHostPort.diValue				:= UINT_TO_DINT(p_tyHermesConfiguration.a_tyUSParam[1].uiHostPort);
	tyP1023McSetHComm.tyUSHermesB.tyStringHostAddr.sValue			:= p_tyHermesConfiguration.a_tyUSParam[1].sHostAddress;
	tyP1023McSetHComm.tyUSHermesB.tyBtnCheckAliveResponse.bValue	:= p_tyHermesConfiguration.a_tyUSParam[1].bFeatureCheckAliveResponse;
	tyP1023McSetHComm.tyUSHermesB.tyBtnCmpTypeId.bValue				:= p_tyHermesConfiguration.a_tyUSParam[1].bCmpTypeId;
	tyP1023McSetHComm.tyUSHermesB.tyBtnCmpParam.bValue				:= p_tyHermesConfiguration.a_tyUSParam[1].bCmpParam;
	tyP1023McSetHComm.tyUSHermesB.tyBtnOverWrite.bValue				:= p_tyHermesConfiguration.a_tyUSParam[1].bOverwrite;
	tyP1023McSetHComm.tyUSHermesB.tyBtnBoardForecast.bValue		:= p_tyHermesConfiguration.a_tyUSParam[0].bFeatureBoardForecast;//new for Hermes 1.3
	tyP1023McSetHComm.tyUSHermesB.tyBtnQueryBoardInfo.bValue		:= p_tyHermesConfiguration.a_tyUSParam[0].bFeatureQueryBoardInfo;//new for Hermes 1.3

	tyP1023McSetHComm.tyUSHermesA.tyBtnBoardForecast.uiRtStat := NOT(p_tyNtParamCurr.bHermesSvyPrep);
	tyP1023McSetHComm.tyUSHermesA.tyBtnQueryBoardInfo.uiRtStat := NOT(p_tyNtParamCurr.bHermesSvyPrep);
	tyP1023McSetHComm.tyUSHermesB.tyBtnBoardForecast.uiRtStat := NOT(p_tyNtParamCurr.bHermesSvyPrep);
	tyP1023McSetHComm.tyUSHermesB.tyBtnQueryBoardInfo.uiRtStat := NOT(p_tyNtParamCurr.bHermesSvyPrep);
END_ACTION
```

#### Act_Main_P1024.st
```iecst
ACTION Act_Main_P1024:

	//Machine Setting - Anti Gap Sensor Filter
	tyP1024McSetAntiGap.tyAntiGap.tyNumLftSenOff.diValueMin	:= p_tyNtParamCurr.tyUIAntiGapSenOffTm.diMin;
	tyP1024McSetAntiGap.tyAntiGap.tyNumLftSenOff.diValueMax	:= p_tyNtParamCurr.tyUIAntiGapSenOffTm.diMax;

	tyP1024McSetAntiGap.tyAntiGap.tyNumMidSenOff.diValueMin	:= p_tyNtParamCurr.tyUIAntiGapSenOffTm.diMin;
	tyP1024McSetAntiGap.tyAntiGap.tyNumMidSenOff.diValueMax	:= p_tyNtParamCurr.tyUIAntiGapSenOffTm.diMax;

	tyP1024McSetAntiGap.tyAntiGap.tyNumRgtSenOff.diValueMin	:= p_tyNtParamCurr.tyUIAntiGapSenOffTm.diMin;
	tyP1024McSetAntiGap.tyAntiGap.tyNumRgtSenOff.diValueMax	:= p_tyNtParamCurr.tyUIAntiGapSenOffTm.diMax;

	tyP1024McSetAntiGap.tyAntiGap.tyNumClrSenOff.diValueMin	:= p_tyNtParamCurr.tyUIAntiGapSenOffTm.diMin;
	tyP1024McSetAntiGap.tyAntiGap.tyNumClrSenOff.diValueMax	:= p_tyNtParamCurr.tyUIAntiGapSenOffTm.diMax;

	tyP1024McSetAntiGap.tyAntiGap.tyNumMagConvEntOff.diValueMin	:= p_tyNtParamCurr.tyUIAntiGapSenOffTm.diMin;
	tyP1024McSetAntiGap.tyAntiGap.tyNumMagConvEntOff.diValueMax	:= p_tyNtParamCurr.tyUIAntiGapSenOffTm.diMax;

	tyP1024McSetAntiGap.tyAntiGap.tyNumMagConvEntOn.diValueMin	:= p_tyNtParamCurr.tyUIAntiGapSenOnTm.diMin;
	tyP1024McSetAntiGap.tyAntiGap.tyNumMagConvEntOn.diValueMax	:= p_tyNtParamCurr.tyUIAntiGapSenOnTm.diMax;

	tyP1024McSetAntiGap.tyAntiGap.tyNumMagConvPresentOff.diValueMin	:= p_tyNtParamCurr.tyUIAntiGapSenOffTm.diMin;
	tyP1024McSetAntiGap.tyAntiGap.tyNumMagConvPresentOff.diValueMax	:= p_tyNtParamCurr.tyUIAntiGapSenOffTm.diMax;

	tyP1024McSetAntiGap.tyAntiGap.tyNumMagConvPresentOn.diValueMin	:= p_tyNtParamCurr.tyUIAntiGapSenOnTm.diMin;
	tyP1024McSetAntiGap.tyAntiGap.tyNumMagConvPresentOn.diValueMax	:= p_tyNtParamCurr.tyUIAntiGapSenOnTm.diMax;

	//Parameter
	tyP1024McSetAntiGap.tyAntiGap.tyNumLftSenOff.diValue	:= p_tyMcParamCurr.tyLftSenAntiGapDly.diSigOffTm;

	tyP1024McSetAntiGap.tyAntiGap.tyNumMidSenOff.diValue	:= p_tyMcParamCurr.tyMidSenAntiGapDly.diSigOffTm;

	tyP1024McSetAntiGap.tyAntiGap.tyNumRgtSenOff.diValue	:= p_tyMcParamCurr.tyRgtSenAntiGapDly.diSigOffTm;

	tyP1024McSetAntiGap.tyAntiGap.tyNumClrSenOff.diValue	:= p_tyMcParamCurr.tyClrSenAntiGapDly.diSigOffTm;

	tyP1024McSetAntiGap.tyAntiGap.tyNumMagConvEntOff.diValue	:= p_tyMcParamCurr.tyMagConvEntrySenAntiGapDly.diSigOffTm;

	tyP1024McSetAntiGap.tyAntiGap.tyNumMagConvEntOn.diValue		:= p_tyMcParamCurr.tyMagConvEntrySenAntiGapDly.diSigOnTm;

	tyP1024McSetAntiGap.tyAntiGap.tyNumMagConvPresentOff.diValue	:= p_tyMcParamCurr.tyMagConvPresentSenAntiGapDly.diSigOffTm;

	tyP1024McSetAntiGap.tyAntiGap.tyNumMagConvPresentOn.diValue		:= p_tyMcParamCurr.tyMagConvPresentSenAntiGapDly.diSigOnTm;

	tyP1024McSetAntiGap.tyAntiGap.tyNumMagConvEntOff.uiRtStat.0 := NOT (p_tyNtParamCurr.bProjMag1ConvPrep AND p_tyNtParamCurr.bProjMag2ConvPrep AND p_tyNtParamCurr.bProjMag3ConvPrep AND p_tyNtParamCurr.bProjLifTravMnlLoad= FALSE);
	tyP1024McSetAntiGap.tyAntiGap.tyNumMagConvEntOn.uiRtStat.0 := NOT (p_tyNtParamCurr.bProjMag1ConvPrep AND p_tyNtParamCurr.bProjMag2ConvPrep AND p_tyNtParamCurr.bProjMag3ConvPrep AND p_tyNtParamCurr.bProjLifTravMnlLoad= FALSE);
	tyP1024McSetAntiGap.tyAntiGap.tyNumMagConvPresentOff.uiRtStat.0 := NOT (p_tyNtParamCurr.bProjMag1ConvPrep AND p_tyNtParamCurr.bProjMag2ConvPrep AND p_tyNtParamCurr.bProjMag3ConvPrep AND p_tyNtParamCurr.bProjLifTravMnlLoad= FALSE);
	tyP1024McSetAntiGap.tyAntiGap.tyNumMagConvPresentOn.uiRtStat.0 := NOT (p_tyNtParamCurr.bProjMag1ConvPrep AND p_tyNtParamCurr.bProjMag2ConvPrep AND p_tyNtParamCurr.bProjMag3ConvPrep AND p_tyNtParamCurr.bProjLifTravMnlLoad= FALSE);

END_ACTION
```

#### Act_Main_P1026.st
```iecst
ACTION Act_Main_P1026:

	//Display
	//Curtain sensor bypass
	IF p_tyNtParamCurr.tyDOSettings.diBypCurtainSen > 0 THEN
		tyP1026McSetTeach.tyTeachLifterPosA.tyBtn4.uiRtStat := FALSE;
		tyP1026McSetTeach.tyTeachLifterPosA.tyBtn4.usiBitmapIdx := 5;
		tyP1026McSetTeach.tyTeachLifterPosA.tyBtn4.usiTxtIdx := 47;
		tyP1026McSetTeach.tyTeachLifterPosB.tyBtn4.uiRtStat := FALSE;
		tyP1026McSetTeach.tyTeachLifterPosB.tyBtn4.usiBitmapIdx := 5;
		tyP1026McSetTeach.tyTeachLifterPosB.tyBtn4.usiTxtIdx := 47;
		tyP1026McSetTeach.tyTeachTravPosA.tyBtn4.uiRtStat := FALSE;
		tyP1026McSetTeach.tyTeachTravPosA.tyBtn4.usiBitmapIdx := 5;
		tyP1026McSetTeach.tyTeachTravPosA.tyBtn4.usiTxtIdx := 47;
		tyP1026McSetTeach.tyTeachTravPosB.tyBtn4.uiRtStat := FALSE;
		tyP1026McSetTeach.tyTeachTravPosB.tyBtn4.usiBitmapIdx := 5;
		tyP1026McSetTeach.tyTeachTravPosB.tyBtn4.usiTxtIdx := 47;
	END_IF

	//Traverser
	tyP1026McSetTeach.tyMotionStdTrav.tyNumTargetPos.diValue		:= 0;
	tyP1026McSetTeach.tyMotionStdTrav.tyNumStepSize.diValue			:= 0;
	tyP1026McSetTeach.tyMotionStdTrav.tyNumNomSpd.diValue			:= (p_tyNtParamCurr.tyUITravNomSpd.diMax + p_tyNtParamCurr.tyUITravNomSpd.diMin) / 2;
	tyP1026McSetTeach.tyMotionStdTrav.tyNumSlwSpd.diValue			:= (p_tyNtParamCurr.tyUITravSlwSpd.diMax + p_tyNtParamCurr.tyUITravSlwSpd.diMin) / 3;

	tyP1026McSetTeach.tyMotionStdTrav.tyNumTargetPos.diValueMax		:= p_tyNtParamCurr.tyUITravTargetPos.diMax;
	tyP1026McSetTeach.tyMotionStdTrav.tyNumTargetPos.diValueMin		:= p_tyNtParamCurr.tyUITravTargetPos.diMin;

	tyP1026McSetTeach.tyMotionStdTrav.tyNumStepSize.diValueMax		:= p_tyNtParamCurr.tyUITravStepSize.diMax;
	tyP1026McSetTeach.tyMotionStdTrav.tyNumStepSize.diValueMin		:= p_tyNtParamCurr.tyUITravStepSize.diMin;

	tyP1026McSetTeach.tyMotionStdTrav.tyNumNomSpd.diValueMax		:= p_tyNtParamCurr.tyUITravNomSpd.diMax;
	tyP1026McSetTeach.tyMotionStdTrav.tyNumNomSpd.diValueMin		:= p_tyNtParamCurr.tyUITravNomSpd.diMin;

	tyP1026McSetTeach.tyMotionStdTrav.tyNumSlwSpd.diValueMax		:= p_tyNtParamCurr.tyUITravSlwSpd.diMax;
	tyP1026McSetTeach.tyMotionStdTrav.tyNumSlwSpd.diValueMin		:= p_tyNtParamCurr.tyUITravSlwSpd.diMin;

	//Lifter
	tyP1026McSetTeach.tyMotionStdLifter.tyNumTargetPos.diValue		:= 0;
	tyP1026McSetTeach.tyMotionStdLifter.tyNumStepSize.diValue		:= 0;
	tyP1026McSetTeach.tyMotionStdLifter.tyNumNomSpd.diValue			:= (p_tyNtParamCurr.tyUILifterNomSpd.diMax + p_tyNtParamCurr.tyUILifterNomSpd.diMin) / 2;
	tyP1026McSetTeach.tyMotionStdLifter.tyNumSlwSpd.diValue			:= (p_tyNtParamCurr.tyUILifterSlwSpd.diMax + p_tyNtParamCurr.tyUILifterSlwSpd.diMin) / 3;

	tyP1026McSetTeach.tyMotionStdLifter.tyNumTargetPos.diValueMax	:= p_tyNtParamCurr.tyUILifterTargetPos.diMax;
	tyP1026McSetTeach.tyMotionStdLifter.tyNumTargetPos.diValueMin	:= p_tyNtParamCurr.tyUILifterTargetPos.diMin;

	tyP1026McSetTeach.tyMotionStdLifter.tyNumStepSize.diValueMax	:= p_tyNtParamCurr.tyUILifterStepSize.diMax;
	tyP1026McSetTeach.tyMotionStdLifter.tyNumStepSize.diValueMin	:= p_tyNtParamCurr.tyUILifterStepSize.diMin;

	tyP1026McSetTeach.tyMotionStdLifter.tyNumNomSpd.diValueMax		:= p_tyNtParamCurr.tyUILifterNomSpd.diMax;
	tyP1026McSetTeach.tyMotionStdLifter.tyNumNomSpd.diValueMin		:= p_tyNtParamCurr.tyUILifterNomSpd.diMin;

	tyP1026McSetTeach.tyMotionStdLifter.tyNumSlwSpd.diValueMax		:= p_tyNtParamCurr.tyUILifterSlwSpd.diMax;
	tyP1026McSetTeach.tyMotionStdLifter.tyNumSlwSpd.diValueMin		:= p_tyNtParamCurr.tyUILifterSlwSpd.diMin;

END_ACTION
```

#### Act_Main_P1027.st
```iecst
ACTION Act_Main_P1027:

	tyP1027McSetOpCon.tyParam.tyNumLineNo.diValue			:= UINT_TO_DINT(p_tyMcParamCurr.tyOpConParam.uiLineNo);
	tyP1027McSetOpCon.tyParam.tyNumStatNo.diValue			:= UINT_TO_DINT(p_tyMcParamCurr.tyOpConParam.uiStatNo);
	tyP1027McSetOpCon.tyParam.tyNumStatIdx.diValue			:= UINT_TO_DINT(p_tyMcParamCurr.tyOpConParam.uiStatIdx);
	tyP1027McSetOpCon.tyParam.tyNumFuNo.diValue				:= UINT_TO_DINT(p_tyMcParamCurr.tyOpConParam.uiFuNo);
	tyP1027McSetOpCon.tyParam.tyNumWorkPos.diValue			:= UINT_TO_DINT(p_tyMcParamCurr.tyOpConParam.uiWorkPos);
	tyP1027McSetOpCon.tyParam.tyNumToolPos.diValue			:= UINT_TO_DINT(p_tyMcParamCurr.tyOpConParam.uiToolPos);
	tyP1027McSetOpCon.tyParam.tyNumProcessNo.diValue		:= UINT_TO_DINT(p_tyMcParamCurr.tyOpConParam.uiProcessNo);
	tyP1027McSetOpCon.tyParam.tyStringProcessNm.sValue		:= p_tyMcParamCurr.tyOpConParam.sProcessName;
	tyP1027McSetOpCon.tyParam.tyStringApplication.sValue	:= p_tyMcParamCurr.tyOpConParam.sApplication;
	tyP1027McSetOpCon.tyParam.tyBtnOpConEn.bValue			:= p_tyMcParamCurr.bOpConEn;
	tyP1027McSetOpCon.tyParam.tyStringOpConSvrIP.sValue		:= p_tyMcParamCurr.sOpConIPAddr;
	tyP1027McSetOpCon.tyParam.tyNumOpConSvrPort.diValue		:= UINT_TO_DINT (p_tyMcParamCurr.uiOpConSvrPort);
END_ACTION
```

#### Act_Main_P1030.st
```iecst
ACTION Act_Main_P1030:

	//P1030 Magazine Settings
	//Display
	tyP1030MagSet.tyMagSet.tyTxtLifMag3Slt1PosLbl.uiRtStat.0	:= NOT(p_tyNtParamCurr.eProjMag = ULMagTriple);
	tyP1030MagSet.tyMagSet.tyNumLifterMag3Slt1Pos.uiRtStat.0	:= NOT(p_tyNtParamCurr.eProjMag = ULMagTriple);
	tyP1030MagSet.tyMagSet.tyBtnLifterMag3Slt1Pos.uiRtStat.0	:= NOT(p_tyNtParamCurr.eProjMag = ULMagTriple);

	tyP1030MagSet.tyMagSet.tyTxtTravPosMag3Lbl.uiRtStat.0	:= NOT(p_tyNtParamCurr.eProjMag = ULMagTriple);
	tyP1030MagSet.tyMagSet.tyNumTravPosMag3.uiRtStat.0		:= NOT(p_tyNtParamCurr.eProjMag = ULMagTriple);
	tyP1030MagSet.tyMagSet.tyBtnTravPosMag3.uiRtStat.0		:= NOT(p_tyNtParamCurr.eProjMag = ULMagTriple);

	tyP1030MagSet.tyMagSet.tyNumSltToSltDist.diValueMin	:= p_tyNtParamCurr.tyUISltToSltDist.diMin;
	tyP1030MagSet.tyMagSet.tyNumSltToSltDist.diValueMax	:= p_tyNtParamCurr.tyUISltToSltDist.diMax;

	tyP1030MagSet.tyMagSet.tyNumMaxSlt.diValueMin	:= p_tyNtParamCurr.diProjMagMinSlt;
	tyP1030MagSet.tyMagSet.tyNumMaxSlt.diValueMax	:= p_tyNtParamCurr.diProjMagMaxSlt;

	tyP1030MagSet.tyMagSet.tyNumLifterMag1Slt1Pos.diValueMin	:= p_tyNtParamCurr.tyUILifterTargetPos.diMin;
	tyP1030MagSet.tyMagSet.tyNumLifterMag1Slt1Pos.diValueMax	:= p_tyNtParamCurr.tyUILifterTargetPos.diMax;
	tyP1030MagSet.tyMagSet.tyNumLifterMag2Slt1Pos.diValueMin	:= p_tyNtParamCurr.tyUILifterTargetPos.diMin;
	tyP1030MagSet.tyMagSet.tyNumLifterMag2Slt1Pos.diValueMax	:= p_tyNtParamCurr.tyUILifterTargetPos.diMax;
	tyP1030MagSet.tyMagSet.tyNumLifterMag3Slt1Pos.diValueMin	:= p_tyNtParamCurr.tyUILifterTargetPos.diMin;
	tyP1030MagSet.tyMagSet.tyNumLifterMag3Slt1Pos.diValueMax	:= p_tyNtParamCurr.tyUILifterTargetPos.diMax;

	tyP1030MagSet.tyMagSet.tyNumTravPosMag1.diValueMin	:= p_tyNtParamCurr.tyUITravTargetPos.diMin;
	tyP1030MagSet.tyMagSet.tyNumTravPosMag1.diValueMax	:= p_tyNtParamCurr.tyUITravTargetPos.diMax;
	tyP1030MagSet.tyMagSet.tyNumTravPosMag2.diValueMin	:= p_tyNtParamCurr.tyUITravTargetPos.diMin;
	tyP1030MagSet.tyMagSet.tyNumTravPosMag2.diValueMax	:= p_tyNtParamCurr.tyUITravTargetPos.diMax;
	tyP1030MagSet.tyMagSet.tyNumTravPosMag3.diValueMin	:= p_tyNtParamCurr.tyUITravTargetPos.diMin;
	tyP1030MagSet.tyMagSet.tyNumTravPosMag3.diValueMax	:= p_tyNtParamCurr.tyUITravTargetPos.diMax;

	FOR i := 1 TO c_uiP1030TableSize DO
		tyP1030MagSet.tyMagSet.tyTableRecipe.a_tyStringDataCol0[i].sValue	:= UINT_TO_STRING(i);
		tyP1030MagSet.tyMagSet.tyTableRecipe.a_tyStringDataCol1[i].sValue	:= p_tyMagRcpCurrList[i].sRcpNm;
		tyP1030MagSet.tyMagSet.tyTableRecipe.a_tyStringDataCol2[i].sValue	:= p_tyMagRcpCurrList[i].sDisplayInfo;
	END_FOR

	tyP1030MagSet.tyMagSet.tyDrpDnMagModel.usiValueMaxIdx	:= 2;

	tyP1030MagSet.tyMagSet.tyNumMagMaxBrdWidth.diValueMin		:= p_tyNtParamCurr.tyProdRcpWidth.diMin;
	tyP1030MagSet.tyMagSet.tyNumMagMaxBrdWidth.diValueMax		:= p_tyNtParamCurr.tyProdRcpWidth.diMax;

	tyP1030MagSet.tyMagSet.tyBtnSafetyBarDisabled.uiRtStat.0 := NOT(p_tyNtParamCurr.bProjMagSafetyBarPrep);

	tyP1030MagSet.tyMagSet.tyBtnMagHeightChkEn.uiRtStat.0	 := NOT(p_tyNtParamCurr.bProjMagHeightChkPrep);

	tyP1030MagSet.tyMagSet.tyBitmapBrder.uiRtStat.0 		 := NOT(p_tyNtParamCurr.bProjMagSafetyBarPrep OR p_tyNtParamCurr.bProjMagHeightChkPrep);

END_ACTION
```

#### Act_Main_P1031.st
```iecst
ACTION Act_Main_P1031:

	//Display
	//Curtain sensor bypass
	IF p_tyNtParamCurr.tyDOSettings.diBypCurtainSen > 0 THEN
		tyP1031MagSetTeach.tyTeachTravPosMag1.tyBtn4.uiRtStat := FALSE;
		tyP1031MagSetTeach.tyTeachTravPosMag1.tyBtn4.usiBitmapIdx := 5;
		tyP1031MagSetTeach.tyTeachTravPosMag1.tyBtn4.usiTxtIdx := 47;
		tyP1031MagSetTeach.tyTeachTravPosMag2.tyBtn4.uiRtStat := FALSE;
		tyP1031MagSetTeach.tyTeachTravPosMag2.tyBtn4.usiBitmapIdx := 5;
		tyP1031MagSetTeach.tyTeachTravPosMag2.tyBtn4.usiTxtIdx := 47;
		tyP1031MagSetTeach.tyTeachTravPosMag3.tyBtn4.uiRtStat := FALSE;
		tyP1031MagSetTeach.tyTeachTravPosMag3.tyBtn4.usiBitmapIdx := 5;
		tyP1031MagSetTeach.tyTeachTravPosMag3.tyBtn4.usiTxtIdx := 47;
		tyP1031MagSetTeach.tyTeachLifterMag1Slt1Pos.tyBtn4.uiRtStat := FALSE;
		tyP1031MagSetTeach.tyTeachLifterMag1Slt1Pos.tyBtn4.usiBitmapIdx := 5;
		tyP1031MagSetTeach.tyTeachLifterMag1Slt1Pos.tyBtn4.usiTxtIdx := 47;
		tyP1031MagSetTeach.tyTeachLifterMag2Slt1Pos.tyBtn4.uiRtStat := FALSE;
		tyP1031MagSetTeach.tyTeachLifterMag2Slt1Pos.tyBtn4.usiBitmapIdx := 5;
		tyP1031MagSetTeach.tyTeachLifterMag2Slt1Pos.tyBtn4.usiTxtIdx := 47;
		tyP1031MagSetTeach.tyTeachLifterMag3Slt1Pos.tyBtn4.uiRtStat := FALSE;
		tyP1031MagSetTeach.tyTeachLifterMag3Slt1Pos.tyBtn4.usiBitmapIdx := 5;
		tyP1031MagSetTeach.tyTeachLifterMag3Slt1Pos.tyBtn4.usiTxtIdx := 47;
	END_IF

	//Traverser
	tyP1031MagSetTeach.tyMotionStdTrav.tyNumTargetPos.diValue		:= 0;
	tyP1031MagSetTeach.tyMotionStdTrav.tyNumStepSize.diValue		:= 0;
	tyP1031MagSetTeach.tyMotionStdTrav.tyNumNomSpd.diValue			:= (p_tyNtParamCurr.tyUITravNomSpd.diMax + p_tyNtParamCurr.tyUITravNomSpd.diMin) / 2;
	tyP1031MagSetTeach.tyMotionStdTrav.tyNumSlwSpd.diValue			:= (p_tyNtParamCurr.tyUITravSlwSpd.diMax + p_tyNtParamCurr.tyUITravSlwSpd.diMin) / 3;

	tyP1031MagSetTeach.tyMotionStdTrav.tyNumTargetPos.diValueMax	:= p_tyNtParamCurr.tyUITravTargetPos.diMax;
	tyP1031MagSetTeach.tyMotionStdTrav.tyNumTargetPos.diValueMin	:= p_tyNtParamCurr.tyUITravTargetPos.diMin;

	tyP1031MagSetTeach.tyMotionStdTrav.tyNumStepSize.diValueMax		:= p_tyNtParamCurr.tyUITravStepSize.diMax;
	tyP1031MagSetTeach.tyMotionStdTrav.tyNumStepSize.diValueMin		:= p_tyNtParamCurr.tyUITravStepSize.diMin;

	tyP1031MagSetTeach.tyMotionStdTrav.tyNumNomSpd.diValueMax		:= p_tyNtParamCurr.tyUITravNomSpd.diMax;
	tyP1031MagSetTeach.tyMotionStdTrav.tyNumNomSpd.diValueMin		:= p_tyNtParamCurr.tyUITravNomSpd.diMin;

	tyP1031MagSetTeach.tyMotionStdTrav.tyNumSlwSpd.diValueMax		:= p_tyNtParamCurr.tyUITravSlwSpd.diMax;
	tyP1031MagSetTeach.tyMotionStdTrav.tyNumSlwSpd.diValueMin		:= p_tyNtParamCurr.tyUITravSlwSpd.diMin;

	//Lifter
	tyP1031MagSetTeach.tyMotionStdLifter.tyNumTargetPos.diValue		:= 0;
	tyP1031MagSetTeach.tyMotionStdLifter.tyNumStepSize.diValue		:= 0;
	tyP1031MagSetTeach.tyMotionStdLifter.tyNumNomSpd.diValue		:= (p_tyNtParamCurr.tyUILifterNomSpd.diMax + p_tyNtParamCurr.tyUILifterNomSpd.diMin) / 2;
	tyP1031MagSetTeach.tyMotionStdLifter.tyNumSlwSpd.diValue		:= (p_tyNtParamCurr.tyUILifterSlwSpd.diMax + p_tyNtParamCurr.tyUILifterSlwSpd.diMin) / 3;

	tyP1031MagSetTeach.tyMotionStdLifter.tyNumTargetPos.diValueMax	:= p_tyNtParamCurr.tyUILifterTargetPos.diMax;
	tyP1031MagSetTeach.tyMotionStdLifter.tyNumTargetPos.diValueMin	:= p_tyNtParamCurr.tyUILifterTargetPos.diMin;

	tyP1031MagSetTeach.tyMotionStdLifter.tyNumStepSize.diValueMax	:= p_tyNtParamCurr.tyUILifterStepSize.diMax;
	tyP1031MagSetTeach.tyMotionStdLifter.tyNumStepSize.diValueMin	:= p_tyNtParamCurr.tyUILifterStepSize.diMin;

	tyP1031MagSetTeach.tyMotionStdLifter.tyNumNomSpd.diValueMax		:= p_tyNtParamCurr.tyUILifterNomSpd.diMax;
	tyP1031MagSetTeach.tyMotionStdLifter.tyNumNomSpd.diValueMin		:= p_tyNtParamCurr.tyUILifterNomSpd.diMin;

	tyP1031MagSetTeach.tyMotionStdLifter.tyNumSlwSpd.diValueMax		:= p_tyNtParamCurr.tyUILifterSlwSpd.diMax;
	tyP1031MagSetTeach.tyMotionStdLifter.tyNumSlwSpd.diValueMin		:= p_tyNtParamCurr.tyUILifterSlwSpd.diMin;

END_ACTION
```

#### Act_Main_P1040.st
```iecst
ACTION Act_Main_P1040:

	//Display
	tyP1040ProdSet.tyProdSet.tyNumProdWidth.diValueMin		:= p_tyNtParamCurr.tyProdRcpWidth.diMin;
	tyP1040ProdSet.tyProdSet.tyNumProdWidth.diValueMax		:= p_tyNtParamCurr.tyProdRcpWidth.diMax;

	tyP1040ProdSet.tyProdSet.tyNumFirstSlt.diValueMin		:= p_tyNtParamCurr.diProjMagMinSlt;

	tyP1040ProdSet.tyProdSet.tyNumPitch.diValueMin			:= p_tyNtParamCurr.tyProdRcpPitch.diMin;

	tyP1040ProdSet.tyProdSet.tyNumBrdPerSlt.diValueMin		:= p_tyNtParamCurr.tyProdRcpBrdPerSlt.diMin;
	tyP1040ProdSet.tyProdSet.tyNumBrdPerSlt.diValueMax		:= p_tyNtParamCurr.tyProdRcpBrdPerSlt.diMax;

	tyP1040ProdSet.tyProdSet.tyNumMinReqFreeBffr.diValueMin	:= p_tyNtParamCurr.tyProdRcpOvenMinReqFreeBffr.diMin;
	tyP1040ProdSet.tyProdSet.tyNumMinReqFreeBffr.diValueMax	:= p_tyNtParamCurr.tyProdRcpOvenMinReqFreeBffr.diMax;

	tyP1040ProdSet.tyProdSet.tyNumBrdPerSlt.uiRtStat.0		:= NOT(p_tyNtParamCurr.bProjBrdPerSltPrep);
	tyP1040ProdSet.tyProdSet.tyTxtBrdPerSlt.uiRtStat.0		:= NOT(p_tyNtParamCurr.bProjBrdPerSltPrep);

	tyP1040ProdSet.tyProdSet.tyNumPshrOffset.uiRtStat.0		:= NOT (p_tyNtParamCurr.bAWPusherPrep);
	tyP1040ProdSet.tyProdSet.tyTxtPshrOffset.uiRtStat.0		:= NOT (p_tyNtParamCurr.bAWPusherPrep);

	//Oven
	tyP1040ProdSet.tyProdSet.tyNumMinReqFreeBffr.uiRtStat.0	:= NOT p_tyNtParamCurr.bOvenInfoPrep;
	tyP1040ProdSet.tyProdSet.tyTxtMinReqFreeBffr.uiRtStat.0	:= NOT p_tyNtParamCurr.bOvenInfoPrep;

	//Machine Mode
	IF p_tyNtParamCurr.bProjLaneBPrep THEN
		tyP1040ProdSet.tyProdSet.tyDrpDnMcMode.usiValueMaxIdx	:= 8;
	ELSE
		tyP1040ProdSet.tyProdSet.tyDrpDnMcMode.usiValueMaxIdx	:= 2;
	END_IF;

	//P1040 Product Settings
	FOR i := 1 TO c_uiP1040TableSize DO
		tyP1040ProdSet.tyProdSet.tyTableRecipe.a_tyStringDataCol0[i].sValue	:= UINT_TO_STRING(i);
		tyP1040ProdSet.tyProdSet.tyTableRecipe.a_tyStringDataCol1[i].sValue	:= p_tyProdRcpCurrList[i].sRcpNm;
		tyP1040ProdSet.tyProdSet.tyTableRecipe.a_tyStringDataCol2[i].sValue	:= p_tyProdRcpCurrList[i].sDisplayInfo;
	END_FOR

	//Motorized Pusher
	tyP1040ProdSet.tyProdSet.tyNumMtrPshrExtSpd.diValueMin	:= p_tyNtParamCurr.tyProdRcpMtrPshrExtSpd.diMin;
	tyP1040ProdSet.tyProdSet.tyNumMtrPshrExtSpd.diValueMax	:= p_tyNtParamCurr.tyProdRcpMtrPshrExtSpd.diMax;

	tyP1040ProdSet.tyProdSet.tyNumMtrPshrExtTorq.diValueMin	:= p_tyNtParamCurr.tyProdRcpMtrPshrExtTorq.diMin;
	tyP1040ProdSet.tyProdSet.tyNumMtrPshrExtTorq.diValueMax	:= p_tyNtParamCurr.tyProdRcpMtrPshrExtTorq.diMax;

	tyP1040ProdSet.tyProdSet.tyNumMtrPshrExtSpd.uiRtStat.0	:= NOT p_tyNtParamCurr.bProjMotorizedPusherPrep;
	tyP1040ProdSet.tyProdSet.tyNumMtrPshrExtTorq.uiRtStat.0	:= NOT p_tyNtParamCurr.bProjMotorizedPusherPrep;

END_ACTION
```

#### Act_Main_P1050.st
```iecst
ACTION Act_Main_P1050:

	//Display
	tyP1050LFSet.tyLdr.tyNumAfterOven.diValueMax	:= p_tyNtParamCurr.tyUILFIndexAfterOven.diMax;
	tyP1050LFSet.tyLdr.tyNumAfterOven.diValueMin	:= p_tyNtParamCurr.tyUILFIndexAfterOven.diMin;
	tyP1050LFSet.tyLdr.tyNumAfterOven2.diValueMax	:= p_tyNtParamCurr.tyUILFIndexAfterOven.diMax;
	tyP1050LFSet.tyLdr.tyNumAfterOven2.diValueMin	:= p_tyNtParamCurr.tyUILFIndexAfterOven.diMin;

	tyP1050LFSet.tyLdr.tyNumBeforeOven.diValueMax	:= p_tyNtParamCurr.tyUILFIndexBeforeOven.diMax;
	tyP1050LFSet.tyLdr.tyNumBeforeOven.diValueMin	:= p_tyNtParamCurr.tyUILFIndexBeforeOven.diMin;
	tyP1050LFSet.tyLdr.tyNumBeforeOven2.diValueMax	:= p_tyNtParamCurr.tyUILFIndexBeforeOven.diMax;
	tyP1050LFSet.tyLdr.tyNumBeforeOven2.diValueMin	:= p_tyNtParamCurr.tyUILFIndexBeforeOven.diMin;

	//Leader
	FOR i := 1 TO c_uiP1050TableSize DO
		tyP1050LFSet.tyLdr.tyTable1List.a_tyStringDataCol2[i].sValue	:= p_tyMcParamCurr.a_sLFIPAddr[i];
		tyP1050LFSet.tyLdr.tyTable1List.a_tyTxtDataCol3[i].usiValueIdx	:= (BOOL_TO_USINT(p_tyMcParamCurr.a_bLFOnline[i])) + 1;
	END_FOR

	//Parameter
	tyP1050LFSet.tyLdr.tyNumAfterOven.diValue	:= p_tyMcParamCurr.diLFMcIdxAfterOven;
	tyP1050LFSet.tyLdr.tyNumBeforeOven.diValue	:= p_tyMcParamCurr.diLFMcIdxBeforeOven;
	tyP1050LFSet.tyLdr.tyNumAfterOven2.diValue	:= p_tyMcParamCurr.diLFMcIdxAfterOven2;
	tyP1050LFSet.tyLdr.tyNumBeforeOven2.diValue	:= p_tyMcParamCurr.diLFMcIdxBeforeOven2;

END_ACTION
```

#### Act_Main_P1080.st
```iecst
ACTION Act_Main_P1080:

	//User Management
	FOR i := 1 TO c_uiP1080TableSize DO
		tyP1080UsrMgmt.tyUsrMgmt.tyTableList.a_tyStringDataCol0[i].sValue		:= UINT_TO_STRING(i);
		tyP1080UsrMgmt.tyUsrMgmt.tyTableList.a_tyStringDataCol1[i].sValue		:= p_tyUsrMgmtAllList[i].sUsrNm;
		tyP1080UsrMgmt.tyUsrMgmt.tyTableList.a_tyTxtDataCol3[i].usiValueIdx		:= DINT_TO_USINT((p_tyUsrMgmtAllList[i].eUsrLvl) + 1);
	END_FOR

END_ACTION
```

#### Act_Main_P1081.st
```iecst
ACTION Act_Main_P1081:

	//User Managment User Access Right
	//Level 1
	IF p_tyUsrMgmtFullData.tyAccessRightLvl1.sNm <> '' THEN
		tyP1081UsrMgmtUsrAccessRgt.tyUsrAccessRgtLvl1.tyStringNm.sValue	:= p_tyUsrMgmtFullData.tyAccessRightLvl1.sNm;
		tyProperty.tyUITxtSnippets.sUsrMgmtUsrLv1Nm						:= p_tyUsrMgmtFullData.tyAccessRightLvl1.sNm;
	ELSE
		tyP1081UsrMgmtUsrAccessRgt.tyUsrAccessRgtLvl1.tyStringNm.sValue	:= tyProperty.tyUITxtSnippets.sUsrMgmtUsrLv1Nm;
	END_IF

	tyP1081UsrMgmtUsrAccessRgt.tyUsrAccessRgtLvl1.tyBtnOps.bValue		:= p_tyUsrMgmtFullData.tyAccessRightLvl1.bOpt;
	tyP1081UsrMgmtUsrAccessRgt.tyUsrAccessRgtLvl1.tyBtnProdSel.bValue	:= p_tyUsrMgmtFullData.tyAccessRightLvl1.bProdSel;
	tyP1081UsrMgmtUsrAccessRgt.tyUsrAccessRgtLvl1.tyBtnMagSel.bValue	:= p_tyUsrMgmtFullData.tyAccessRightLvl1.bMagSel;
	tyP1081UsrMgmtUsrAccessRgt.tyUsrAccessRgtLvl1.tyBtnMcInfo.bValue	:= p_tyUsrMgmtFullData.tyAccessRightLvl1.bMcInfo;
	tyP1081UsrMgmtUsrAccessRgt.tyUsrAccessRgtLvl1.tyBtnAlm.bValue		:= p_tyUsrMgmtFullData.tyAccessRightLvl1.bAlm;
	tyP1081UsrMgmtUsrAccessRgt.tyUsrAccessRgtLvl1.tyBtnBffrInfo.bValue	:= p_tyUsrMgmtFullData.tyAccessRightLvl1.bBffrInfo;
	tyP1081UsrMgmtUsrAccessRgt.tyUsrAccessRgtLvl1.tyBtnOvenInfo.bValue	:= p_tyUsrMgmtFullData.tyAccessRightLvl1.bOvenInfo;
	tyP1081UsrMgmtUsrAccessRgt.tyUsrAccessRgtLvl1.tyBtnMagInfo.bValue	:= p_tyUsrMgmtFullData.tyAccessRightLvl1.bMagInfo;
	tyP1081UsrMgmtUsrAccessRgt.tyUsrAccessRgtLvl1.tyBtnLFCtrl.bValue	:= p_tyUsrMgmtFullData.tyAccessRightLvl1.bLFCtrl;
	tyP1081UsrMgmtUsrAccessRgt.tyUsrAccessRgtLvl1.tyBtnManual.bValue	:= p_tyUsrMgmtFullData.tyAccessRightLvl1.bManual;
	tyP1081UsrMgmtUsrAccessRgt.tyUsrAccessRgtLvl1.tyBtnSimu.bValue		:= p_tyUsrMgmtFullData.tyAccessRightLvl1.bSimulation;
	tyP1081UsrMgmtUsrAccessRgt.tyUsrAccessRgtLvl1.tyBtnProdSet.bValue	:= p_tyUsrMgmtFullData.tyAccessRightLvl1.bProdSet;
	tyP1081UsrMgmtUsrAccessRgt.tyUsrAccessRgtLvl1.tyBtnMagSet.bValue	:= p_tyUsrMgmtFullData.tyAccessRightLvl1.bMagSet;
	tyP1081UsrMgmtUsrAccessRgt.tyUsrAccessRgtLvl1.tyBtnMcSet.bValue		:= p_tyUsrMgmtFullData.tyAccessRightLvl1.bMcSet;
	tyP1081UsrMgmtUsrAccessRgt.tyUsrAccessRgtLvl1.tyBtnLang.bValue		:= p_tyUsrMgmtFullData.tyAccessRightLvl1.bLang;
	tyP1081UsrMgmtUsrAccessRgt.tyUsrAccessRgtLvl1.tyBtnLFSet.bValue		:= p_tyUsrMgmtFullData.tyAccessRightLvl1.bLFSet;
	tyP1081UsrMgmtUsrAccessRgt.tyUsrAccessRgtLvl1.tyBtnChgParam.bValue	:= p_tyUsrMgmtFullData.tyAccessRightLvl1.bChgParam;

	//Level 2
	IF p_tyUsrMgmtFullData.tyAccessRightLvl2.sNm <> '' THEN
		tyP1081UsrMgmtUsrAccessRgt.tyUsrAccessRgtLvl2.tyStringNm.sValue	:= p_tyUsrMgmtFullData.tyAccessRightLvl2.sNm;
		tyProperty.tyUITxtSnippets.sUsrMgmtUsrLv2Nm						:= p_tyUsrMgmtFullData.tyAccessRightLvl2.sNm;
	ELSE
		tyP1081UsrMgmtUsrAccessRgt.tyUsrAccessRgtLvl2.tyStringNm.sValue	:= tyProperty.tyUITxtSnippets.sUsrMgmtUsrLv2Nm;
	END_IF

	tyP1081UsrMgmtUsrAccessRgt.tyUsrAccessRgtLvl2.tyBtnOps.bValue		:= p_tyUsrMgmtFullData.tyAccessRightLvl2.bOpt;
	tyP1081UsrMgmtUsrAccessRgt.tyUsrAccessRgtLvl2.tyBtnProdSel.bValue	:= p_tyUsrMgmtFullData.tyAccessRightLvl2.bProdSel;
	tyP1081UsrMgmtUsrAccessRgt.tyUsrAccessRgtLvl2.tyBtnMagSel.bValue	:= p_tyUsrMgmtFullData.tyAccessRightLvl2.bMagSel;
	tyP1081UsrMgmtUsrAccessRgt.tyUsrAccessRgtLvl2.tyBtnMcInfo.bValue	:= p_tyUsrMgmtFullData.tyAccessRightLvl2.bMcInfo;
	tyP1081UsrMgmtUsrAccessRgt.tyUsrAccessRgtLvl2.tyBtnAlm.bValue		:= p_tyUsrMgmtFullData.tyAccessRightLvl2.bAlm;
	tyP1081UsrMgmtUsrAccessRgt.tyUsrAccessRgtLvl2.tyBtnBffrInfo.bValue	:= p_tyUsrMgmtFullData.tyAccessRightLvl2.bBffrInfo;
	tyP1081UsrMgmtUsrAccessRgt.tyUsrAccessRgtLvl2.tyBtnOvenInfo.bValue	:= p_tyUsrMgmtFullData.tyAccessRightLvl2.bOvenInfo;
	tyP1081UsrMgmtUsrAccessRgt.tyUsrAccessRgtLvl2.tyBtnMagInfo.bValue	:= p_tyUsrMgmtFullData.tyAccessRightLvl2.bMagInfo;
	tyP1081UsrMgmtUsrAccessRgt.tyUsrAccessRgtLvl2.tyBtnLFCtrl.bValue	:= p_tyUsrMgmtFullData.tyAccessRightLvl2.bLFCtrl;
	tyP1081UsrMgmtUsrAccessRgt.tyUsrAccessRgtLvl2.tyBtnManual.bValue	:= p_tyUsrMgmtFullData.tyAccessRightLvl2.bManual;
	tyP1081UsrMgmtUsrAccessRgt.tyUsrAccessRgtLvl2.tyBtnSimu.bValue		:= p_tyUsrMgmtFullData.tyAccessRightLvl2.bSimulation;
	tyP1081UsrMgmtUsrAccessRgt.tyUsrAccessRgtLvl2.tyBtnProdSet.bValue	:= p_tyUsrMgmtFullData.tyAccessRightLvl2.bProdSet;
	tyP1081UsrMgmtUsrAccessRgt.tyUsrAccessRgtLvl2.tyBtnMagSet.bValue	:= p_tyUsrMgmtFullData.tyAccessRightLvl2.bMagSet;
	tyP1081UsrMgmtUsrAccessRgt.tyUsrAccessRgtLvl2.tyBtnMcSet.bValue		:= p_tyUsrMgmtFullData.tyAccessRightLvl2.bMcSet;
	tyP1081UsrMgmtUsrAccessRgt.tyUsrAccessRgtLvl2.tyBtnLang.bValue		:= p_tyUsrMgmtFullData.tyAccessRightLvl2.bLang;
	tyP1081UsrMgmtUsrAccessRgt.tyUsrAccessRgtLvl2.tyBtnLFSet.bValue		:= p_tyUsrMgmtFullData.tyAccessRightLvl2.bLFSet;
	tyP1081UsrMgmtUsrAccessRgt.tyUsrAccessRgtLvl2.tyBtnChgParam.bValue	:= p_tyUsrMgmtFullData.tyAccessRightLvl2.bChgParam;

	//Level 3
	IF p_tyUsrMgmtFullData.tyAccessRightLvl3.sNm <> '' THEN
		tyP1081UsrMgmtUsrAccessRgt.tyUsrAccessRgtLvl3.tyStringNm.sValue	:= p_tyUsrMgmtFullData.tyAccessRightLvl3.sNm;
		tyProperty.tyUITxtSnippets.sUsrMgmtUsrLv3Nm						:= p_tyUsrMgmtFullData.tyAccessRightLvl3.sNm;
	ELSE
		tyP1081UsrMgmtUsrAccessRgt.tyUsrAccessRgtLvl3.tyStringNm.sValue	:= tyProperty.tyUITxtSnippets.sUsrMgmtUsrLv3Nm;
	END_IF

	tyP1081UsrMgmtUsrAccessRgt.tyUsrAccessRgtLvl3.tyBtnOps.bValue		:= p_tyUsrMgmtFullData.tyAccessRightLvl3.bOpt;
	tyP1081UsrMgmtUsrAccessRgt.tyUsrAccessRgtLvl3.tyBtnProdSel.bValue	:= p_tyUsrMgmtFullData.tyAccessRightLvl3.bProdSel;
	tyP1081UsrMgmtUsrAccessRgt.tyUsrAccessRgtLvl3.tyBtnMagSel.bValue	:= p_tyUsrMgmtFullData.tyAccessRightLvl3.bMagSel;
	tyP1081UsrMgmtUsrAccessRgt.tyUsrAccessRgtLvl3.tyBtnMcInfo.bValue	:= p_tyUsrMgmtFullData.tyAccessRightLvl3.bMcInfo;
	tyP1081UsrMgmtUsrAccessRgt.tyUsrAccessRgtLvl3.tyBtnAlm.bValue		:= p_tyUsrMgmtFullData.tyAccessRightLvl3.bAlm;
	tyP1081UsrMgmtUsrAccessRgt.tyUsrAccessRgtLvl3.tyBtnBffrInfo.bValue	:= p_tyUsrMgmtFullData.tyAccessRightLvl3.bBffrInfo;
	tyP1081UsrMgmtUsrAccessRgt.tyUsrAccessRgtLvl3.tyBtnOvenInfo.bValue	:= p_tyUsrMgmtFullData.tyAccessRightLvl3.bOvenInfo;
	tyP1081UsrMgmtUsrAccessRgt.tyUsrAccessRgtLvl3.tyBtnMagInfo.bValue	:= p_tyUsrMgmtFullData.tyAccessRightLvl3.bMagInfo;
	tyP1081UsrMgmtUsrAccessRgt.tyUsrAccessRgtLvl3.tyBtnLFCtrl.bValue	:= p_tyUsrMgmtFullData.tyAccessRightLvl3.bLFCtrl;
	tyP1081UsrMgmtUsrAccessRgt.tyUsrAccessRgtLvl3.tyBtnManual.bValue	:= p_tyUsrMgmtFullData.tyAccessRightLvl3.bManual;
	tyP1081UsrMgmtUsrAccessRgt.tyUsrAccessRgtLvl3.tyBtnSimu.bValue		:= p_tyUsrMgmtFullData.tyAccessRightLvl3.bSimulation;
	tyP1081UsrMgmtUsrAccessRgt.tyUsrAccessRgtLvl3.tyBtnProdSet.bValue	:= p_tyUsrMgmtFullData.tyAccessRightLvl3.bProdSet;
	tyP1081UsrMgmtUsrAccessRgt.tyUsrAccessRgtLvl3.tyBtnMagSet.bValue	:= p_tyUsrMgmtFullData.tyAccessRightLvl3.bMagSet;
	tyP1081UsrMgmtUsrAccessRgt.tyUsrAccessRgtLvl3.tyBtnMcSet.bValue		:= p_tyUsrMgmtFullData.tyAccessRightLvl3.bMcSet;
	tyP1081UsrMgmtUsrAccessRgt.tyUsrAccessRgtLvl3.tyBtnLang.bValue		:= p_tyUsrMgmtFullData.tyAccessRightLvl3.bLang;
	tyP1081UsrMgmtUsrAccessRgt.tyUsrAccessRgtLvl3.tyBtnLFSet.bValue		:= p_tyUsrMgmtFullData.tyAccessRightLvl3.bLFSet;
	tyP1081UsrMgmtUsrAccessRgt.tyUsrAccessRgtLvl3.tyBtnChgParam.bValue	:= p_tyUsrMgmtFullData.tyAccessRightLvl3.bChgParam;

END_ACTION
```

#### Package Logical/UI/UI/Act_Background - Change By Project

#### Act_ChgPage.st
```iecst
ACTION Act_ChgPage:

	(*Exit Page*)
	IF (eChgPage <> eChgPageOld) OR (usiChgPage = 2) AND p_bStartupRun = FALSE THEN

		usiChgPage	:= 2;

		CASE eChgPageOld OF

			UIP0700LFCtrl:
				Act_ExitP0700;

			UIP1000Lang:
				Act_ExitP1000;

			UIP1021McSetGen:
				Act_ExitP1021;

			UIP1022McSetVComm:
				Act_ExitP1022;

			UIP1023McSetHComm:
				Act_ExitP1023;

			UIP1024McSetAntiGap:
				Act_ExitP1024;

			UIP1025McSetScan:
				Act_ExitP1025;

			UIP1026McSetTeach:
				Act_ExitP1026;

			UIP1027McSetOpCon:
				Act_ExitP1027;

			UIP1031MagSetTeach:
				Act_ExitP1031;

			UIP1080UsrMgmt:
				Act_ExitP1080;

			UIP1081UsrMgmtUsrAccessRgt:
				Act_ExitP1081;

			ELSE
				usiChgPage	:= 1;

		END_CASE

		IF usiChgPage = 1 THEN
			eChgPageOld		:= eChgPage;
		END_IF

	(*Enter Page*)
	ELSIF usiChgPage = 1 THEN

		CASE eChgPage OF

			UIP0001Startup:
				Act_EntP0001Disp;

			UIP0002Menu:
				Act_EntP0002Disp;

			UIP0003MMenu:
				Act_EntP0003Disp;

			UIP0100Login:
				Act_EntP0100Disp;

			UIP0200OpsGen:
				Act_EntP0200Disp;

			UIP0201OpsTravLifter:
				Act_EntP0201Disp;

			UIP0202OpsMag1:
				Act_EntP0202Disp;

			UIP0203OpsMag2:
				Act_EntP0203Disp;

			UIP0204OpsMag3:
				Act_EntP0204Disp;

			UIP0205OpsAIV:
				Act_EntP0205Disp;

			UIP0206OpsMagConv1:
				Act_EntP0206Disp;

			UIP0207OpsMagConv2:
				Act_EntP0207Disp;

			UIP0300McInfo:
				Act_EntP0300Disp;

			UIP0400ProdSel:
				Act_EntP0400Disp;

			UIP0410MagSel:
				Act_EntP0410Disp;

			UIP0600Alm:
				Act_EntP0600Disp;

			UIP0700LFCtrl:
				Act_EntP0700Disp;

			UIP0800MagInfo:
				Act_EntP0800Disp;

			UIP0850OvenInfo:
				Act_EntP0850Disp;

			UIP0900GenIn:
				Act_EntP0900Disp;

			UIP0910GenOut:
				Act_EntP0910Disp;

			UIP0920MtrNPneuCtrl:
				Act_EntP0920Disp;

			UIP0921Shutter:
				Act_EntP0921Disp;

			UIP0922Stopper:
				Act_EntP0922Disp;

			UIP0923SafetyBar:
				Act_EntP0923Disp;

			UIP0926LifterConv:
				Act_EntP0926Disp;

			UIP0927LifterConv2:
				Act_EntP0927Disp;

			UIP0928MagConv:
				Act_EntP0928Disp;

			UIP0929MagConv2:
				Act_EntP0929Disp;

			UIP0930MagConv1:
				Act_EntP0930Disp;

			UIP0931MagConv2:
				Act_EntP0931Disp;

			UIP0932MagConv3:
				Act_EntP0932Disp;

			UIP0933PusherConv:
				Act_EntP0933Disp;

			UIP0934AW:
				Act_EntP0934Disp;

			UIP0935Lifter:
				Act_EntP0935Disp;

			UIP0936Trav:
				Act_EntP0936Disp;

			UIP0937AWPushOrPuller:
				Act_EntP0937Disp;

			UIP0938MagAW:
				Act_EntP0938Disp;

			UIP0939Lifter2:
				Act_EntP0939Disp;

			UIP0940CommCtrl:
				Act_EntP0940Disp;

			UIP0950Simu:
				Act_EntP0950Disp;

			UIP1000Lang:
				Act_EntP1000Disp;

			UIP1020McSetNavi:
				Act_EntP1020Disp;

			UIP1021McSetGen:
				Act_EntP1021Disp;

			UIP1022McSetVComm:
				Act_EntP1022Disp;

			UIP1023McSetHComm:
				Act_EntP1023Disp;

			UIP1024McSetAntiGap:
				Act_EntP1024Disp;

			UIP1025McSetScan:
				Act_EntP1025Disp;

			UIP1026McSetTeach:
				Act_EntP1026Disp;

			UIP1027McSetOpCon:
				Act_EntP1027Disp;

			UIP1030MagSet:
				Act_EntP1030Disp;

			UIP1031MagSetTeach:
				Act_EntP1031Disp;

			UIP1040ProdSet:
				Act_EntP1040Disp;

			UIP1050LFSet:
				Act_EntP1050Disp;

			UIP1080UsrMgmt:
				Act_EntP1080Disp;

			UIP1081UsrMgmtUsrAccessRgt:
				Act_EntP1081Disp;

		END_CASE

		usiChgPage	:= 0;

		tyProperty.tyVisu.uiChgPage	:= UDINT_TO_UINT(eChgPage);

	END_IF

END_ACTION
```
